// TwinCAT 3 PLC project TcoIoTests
// Title: TcoIoTests
// Company: Vortex.Library
// ProjectVersion: 1.19.1.1780
// ProgramVersion: 3.1.4024.12
// libraries:
//   Tc2_Standard, * (Beckhoff Automation GmbH)
//   Tc2_System, * (Beckhoff Automation GmbH)
//   Tc3_Module, * (Beckhoff Automation GmbH)
//   TcoCore, 0.6.0.913 (Vortex.Library)
//   TcoIo, 0.6.0.913 (Vortex.Library)
// project tree:
//   / PlcTask.TcTTO
//   POUs/ MAIN.TcPOU, tcc.TcPOU, TestEcatComponent.TcPOU
//   DUTs/IO/PdoEntries/ Status_3D84275F.TcDUT, Ctrl_1EFB4D3B.TcDUT, Ctrl_71604E86.TcDUT, Status_B0753356.TcDUT, Status_F2CE6D91.TcDUT, U1_Status_DC903920.TcDUT, U1_Samples_25492287.TcDUT, I1_Status_DC903920.TcDUT, I1_Samples_25492287.TcDUT, U2_Status_DC903920.TcDUT, U2_Samples_25492287.TcDUT, I2_Status_DC903920.TcDUT, I2_Samples_25492287.TcDUT, U3_Status_DC903920.TcDUT, U3_Samples_25492287.TcDUT, I3_Status_DC903920.TcDUT, I3_Samples_25492287.TcDUT, StartTimeNextLatch_02E0C1C8.TcDUT, Status_642C2ED1.TcDUT, Ctrl_77460BD3.TcDUT, Outputs_A910484D.TcDUT, Status_B6795845.TcDUT, Control_C948E0F2.TcDUT, Status_439F40C3.TcDUT, Settings_24C04940.TcDUT, Control_E49DBA1B.TcDUT, Status_8CBE219F.TcDUT, Control_6EF2C5D0.TcDUT
//   DUTs/IO/PDOs/ COM_TxPDO_Map_Inputs_Channel_3801C95E.TcDUT, COM_RxPDO_Map_Outputs_Channel_EADA2E0D.TcDUT, Channel_830843C1.TcDUT, Channel_42CA91F7.TcDUT, AO_Output_Channel_BA7EBB7C.TcDUT, COM_Inputs_3801C95E.TcDUT, COM_Outputs_DEF408EC.TcDUT, AI_Standard_Channel_A8DF64E3.TcDUT, AI_Standard_Channel_4A394481.TcDUT, L1_Voltage_Status_7371B043.TcDUT, L1_Voltage_Samples_41AEB7FF.TcDUT, L1_Current_Status_82DECBF6.TcDUT, L1_Current_Samples_9EC08B3E.TcDUT, L2_Voltage_Status_0D1813FE.TcDUT, L2_Voltage_Samples_75D833AF.TcDUT, L2_Current_Status_FCB7684B.TcDUT, L2_Current_Samples_AAB60F6E.TcDUT, L3_Voltage_Status_273F7295.TcDUT, L3_Voltage_Samples_660A4F9F.TcDUT, L3_Current_Status_D6900920.TcDUT, L3_Current_Samples_B964735E.TcDUT, AI_NextSync1Time_6DC4D296.TcDUT, AI_Sample_Count_EA88CAD9.TcDUT, InfoData_B84DBEC5.TcDUT, MTO_Inputs_Channel_53C09E8B.TcDUT, MTO_Outputs_10x_Channel_A3C0C022.TcDUT, PM_Inputs_Channel_2F868086.TcDUT, PM_Status_data_2A9514CB.TcDUT, PM_Outputs_Channel_E5FBDE30.TcDUT, AT_x_4EC2E768.TcDUT, MDT_864618EC.TcDUT, InfoData_F60A43AC.TcDUT, Device_State_B9CC7757.TcDUT, Device_Control_33EFE70E.TcDUT, Inputs_03C60166.TcDUT, Outputs_79BC345B.TcDUT, Module_1_32_Byte_Valve_Unit_0x7F_1A3DA03C.TcDUT, InfoData_8F85596B.TcDUT, Device_State_384275F8.TcDUT, Device_Control_5857DF0F.TcDUT, Inputs_23559BB0.TcDUT, Outputs_FC2FACAD.TcDUT, Module_1_32_Byte_Valve_Unit_0x7F_85784B27.TcDUT, DI_TxPDO_Map_DF955083.TcDUT, DO_RxPDO_Map_8BCFF4C9.TcDUT, DCM_Status_Channel_36ED096F.TcDUT, DCM_Synchron_info_data_Channel_6FB37C88.TcDUT, DCM_Control_Channel_5A8B5016.TcDUT, DCM_Velocity_Channel_A47A3F41.TcDUT, InfoData_F38373C9.TcDUT, Inputs_424E3ECB.TcDUT, Inputs_84513182.TcDUT, Outputs_3179CEF4.TcDUT, NewMessageFlag_557A079F.TcDUT, Gateway_to_EtherCAT_Data_100_Bytes_AE1F4D6F.TcDUT, EtherCAT_to_Gateway_Data_100_Bytes_44CA1D22.TcDUT, FB_Position_3FA094ED.TcDUT, DRV_Statusword_9B36FDFC.TcDUT, DRV_Following_error_actual_value_5AA320BF.TcDUT, DRV_Controlword_F3F14721.TcDUT, DRV_Target_position_05240F14.TcDUT, InfoData_433F0777.TcDUT, SAI_Inputs_Channel_9DCD6557.TcDUT, SAI_Range_Channel_BDBF6DA9.TcDUT, SAI_Inputs_Real_Channel_CCECF13D.TcDUT, SAI_Range_Control_Channel_F5D9BC22.TcDUT, In_389F2F15.TcDUT, Out_81AAEF2D.TcDUT, ENC_Status_compact_4D066E1A.TcDUT, STM_Status_36ED096F.TcDUT, ENC_Control_compact_21E2D14D.TcDUT, STM_Control_5A8B5016.TcDUT, STM_Velocity_A47A3F41.TcDUT, InfoData_D50C8545.TcDUT, AT_x_26CC547D.TcDUT
//   DUTs/IO/Boxes/ EK1200_013D0B49.TcDUT, EL6002_CD897635.TcDUT, EL1809_32157CFD.TcDUT, EL2809_2B6483BD.TcDUT, EL4004_E203F875.TcDUT, EL6001_0DE01E7E.TcDUT, EL9011_D65D3D32.TcDUT, EK1100_1FC0878B.TcDUT, EK1122_1FC0878B.TcDUT, EL3174_B71BFF42.TcDUT, EL3011_7A495228.TcDUT, EL2008_E2806B95.TcDUT, EK1110_1FC0878B.TcDUT, EL1819_32157CFD.TcDUT, EL2788_E2806B95.TcDUT, EL3773_F128CC82.TcDUT, EL2258_E3B260FA.TcDUT, EL3164_B71BFF42.TcDUT, EL3403_812980A6.TcDUT, EL3024_C6E76B5A.TcDUT, AX5101_1BD22F51.TcDUT, AX5106_1BD22F51.TcDUT, AES_A3B07071.TcDUT, EL6631_A0EC075C.TcDUT, EL9010_D29C2085.TcDUT, AES_B47A2610.TcDUT, IMecat_x_75C6CB6B.TcDUT, AX5103_1BD22F51.TcDUT, EL7332_DFB2BED7.TcDUT, CMMP_93B92D52.TcDUT, Flexi_Gateway_GETC1_429ECB70.TcDUT, EL7211_008D5C9A.TcDUT, EL3692_73B94100.TcDUT, EPP1322_1FC0878B.TcDUT, EPP1008_78E8D3DD.TcDUT, EPP1332_1FC0878B.TcDUT, Flexi_Soft_EtherCAT_Gateway_DE394EDD.TcDUT, EL7041_86DE63E7.TcDUT, IndraDrive_MPB20_C66205C3.TcDUT, EPP2308_F6D9A8D1.TcDUT
//   DUTs/IO/Devices/ SyncUnitTasks_5FDC9770.TcDUT, SyncUnits_C3A34B50.TcDUT, SyncUnits_F0D163CC.TcDUT, SyncUnits_5BE71B8B.TcDUT
//   DUTs/IO/Topology/ Term_1_EK1200_B38DC9A8.TcDUT, Device_1_EtherCAT_49C09C66.TcDUT, Term_11_EK1100_B6553301.TcDUT, Term_18_EK1100_20659A8D.TcDUT, Term_25_EK1100_08217EB4.TcDUT, Term_28_EK1100_415F4A7E.TcDUT, Term_24_EK1122_39E7B5CB.TcDUT, Term_23_EK1100_DFBF0BE4.TcDUT, Term_10_EK1122_3D069EC1.TcDUT, Term_9_EK1100_91BFEC25.TcDUT, Device_2_EtherCAT_22CD061B.TcDUT, Term_157_EK1100_7C4BDD77.TcDUT, Term_158_EK1100_E3D699B1.TcDUT, Term_154_EK1122_E57516AE.TcDUT, Term_153_EK1100_91C0BB48.TcDUT, Term_180_EK1100_796B7783.TcDUT, Term_182_EK1100_E6B2C35E.TcDUT, Term_179_EK1122_2A33725A.TcDUT, Term_178_EK1100_9B7E9852.TcDUT, Term_147_EK1122_CA6A5D16.TcDUT, Term_189_EK1100_06A16014.TcDUT, Term_194_EK1100_D4E2C05F.TcDUT, Term_188_EK1122_78D8AA43.TcDUT, Term_187_EK1100_648C31BD.TcDUT, Term_231_EK1100_6FCE8CEB.TcDUT, Term_233_EK1100_CB654C3B.TcDUT, Term_230_EK1122_16418046.TcDUT, Term_207_EK1100_2D36550A.TcDUT, Term_186_EK1122_75C79D52.TcDUT, Term_237_EK1122_86A8F7BD.TcDUT, Term_289_EK1100_9C677E50.TcDUT, Term_294_EK1100_DFE2A59E.TcDUT, Term_331_EK1100_B9C4E092.TcDUT, Term_333_EK1100_1D6F2042.TcDUT, Term_330_EK1122_0EDE60FE.TcDUT, Term_307_EK1100_EB8FAA41.TcDUT, Term_288_EK1122_18F8921F.TcDUT, Term_146_EK1100_439F5464.TcDUT, Device_3_EtherCAT_368E547E.TcDUT, R1_A2_EC_EK1122_F4361AFD.TcDUT, R1_A3_EC_EK1122_981C12E1.TcDUT, R1_A4_X1_EK1100_C601B400.TcDUT, R1_A4_X2_A2_EK1122_39ABCC27.TcDUT, R1_A4_X2_EK1100_6F5FB3BA.TcDUT, R1_A4_EC_EK1122_467C5A0B.TcDUT, R1_EK1100_4AD22B7B.TcDUT, R2_A2_EC_EK1122_6D3594D4.TcDUT, R2_EK1100_10D8A594.TcDUT, R3_A2_EC_EK1122_9D59CDC8.TcDUT, R3_EK1100_C7887D6C.TcDUT, RH_A2_X2_EK1100_67419BB1.TcDUT, RH_A2_EK1122_10728E09.TcDUT, RH_EK1100_A5940DFE.TcDUT, R4_A2_EC_EK1122_254454A1.TcDUT, R4_EK1100_46A1248C.TcDUT, A2_EK1122_967E4A9C.TcDUT, R4A_EK1100_48316913.TcDUT, R5_A2_EC_EK1122_D562526C.TcDUT, R5_EK1100_0007A337.TcDUT, R6_EK1100_8C41F5F2.TcDUT, R7_A2_EC_EK1122_B7F046E4.TcDUT, R7_EK1100_F50DDAC8.TcDUT, R8_AB0_EPP1322_0001_1BB6BCA8.TcDUT, R8_A2_EK1122_E74C4B62.TcDUT, R8_A3_EK1122_71CA94BA.TcDUT, RC10_A2_EK1122_BBB6F36B.TcDUT, RC10_EPP_EPP1322_0001_810E0540.TcDUT, RC10_A3_EK1122_A50FC1ED.TcDUT, RC10_1_EK1100_40BAEC0F.TcDUT, RC10_2_EK1100_27865421.TcDUT, RC20_A2_EK1122_77321D67.TcDUT, RC20_EPP_EPP1322_0001_59D450BA.TcDUT, RC20_A3_EK1122_1263CE61.TcDUT, RC20_1_EK1100_F221D0A9.TcDUT, RC20_2_EK1100_5EABB509.TcDUT, R8_A8_EK1122_2533F93A.TcDUT, RC30_A2_EK1122_334E4763.TcDUT, RC30_EPP_EPP1322_0001_EDDD6881.TcDUT, RC30_A3_EK1122_482A08F6.TcDUT, RC30_1_EK1100_B995809E.TcDUT, RC30_2_EK1100_8A0FE17C.TcDUT, RC40_A2_EK1122_EAFADCC8.TcDUT, RC40_EPP_EPP1322_0001_ECA1E6F9.TcDUT, RC40_A3_EK1122_E505EE87.TcDUT, RC40_1_EK1100_B918F64D.TcDUT, RC40_2_EK1100_ACF07759.TcDUT, R8_A9_EK1122_3EDD8752.TcDUT, RC50_A2_EK1122_AE8686CC.TcDUT, RC50_EPP_EPP1322_0001_58A8DEC2.TcDUT, RC50_A3_EK1122_7F1D927D.TcDUT, RC50_1_EK1100_D6E64946.TcDUT, RC50_2_EK1100_7854232C.TcDUT, RC60_A2_EK1122_620268C0.TcDUT, RC60_EPP_EPP1322_0001_80728B38.TcDUT, RC60_A3_EK1122_0BEA55B5.TcDUT, RC60_1_EK1100_9BABA6E0.TcDUT, RC60_2_EK1100_0179C204.TcDUT, R8_A10_EK1122_484442E0.TcDUT, RC70_A2_EK1122_267E32C4.TcDUT, RC70_EPP_EPP1322_0001_347BB303.TcDUT, RC70_A3_EK1122_27C9256F.TcDUT, RC70_1_EK1100_B905944A.TcDUT, RC70_2_EK1100_D5DD9671.TcDUT, RC80_A2_EK1122_C3467012.TcDUT, RC80_EPP_EPP1322_0001_828B97C8.TcDUT, RC80_A3_EK1122_B1484BA9.TcDUT, RC80_1_EK1100_5DD08FF5.TcDUT, RC80_2_EK1100_DC1461B5.TcDUT, R8_A11_EK1122_3ED7E2A8.TcDUT, RP10_A2_EK1122_55AC9C5A.TcDUT, RP10_EK1100_26DB4001.TcDUT, RP20_A2_EK1122_68D808EA.TcDUT, RP20_EK1100_7A23D5FF.TcDUT, R8_A12_EK1122_5B843125.TcDUT, RP30_A2_EK1122_C3CC9CB4.TcDUT, RP30_EK1100_66AE6AB6.TcDUT, R8_A13_EK1122_C6957FFB.TcDUT, R8_EK1100_9C7B3B67.TcDUT, R9_AB0_EPP1322_0001_BD7A28FA.TcDUT, R9_A2_EK1122_81F50509.TcDUT, R9_A3_EK1122_C18C26F5.TcDUT, R9_EK1100_484053C0.TcDUT, R10_A2_EK1122_75D61001.TcDUT, R10_AB01_EPP1332_0001_D97A7767.TcDUT, R10_AB00_EPP1322_0001_481BC624.TcDUT, R10_A3_EK1122_6A26DC25.TcDUT, R10_EK1100_C5CE1D87.TcDUT, Device_4_EtherCAT_07442C6B.TcDUT, Term_279_EK1100_ED7D6272.TcDUT, Term_554_EK1100_B580E218.TcDUT, Term_748_EK1100_BC4343B1.TcDUT, Term_881_EK1100_F732F370.TcDUT, Term_1047_EK1100_7ACEE53D.TcDUT, Device_5_EtherCAT_0A694E3C.TcDUT
//   GVLs/ GVL_iXlinker.TcGVL
// (motion and I/O tree: see PLC project tcoio)
// real-time tasks:
//   TASK PlcTask: cycle T#10ms, priority 20, ADS port 350
//   TASK PlcTask1: cycle T#10ms, priority 21, ADS port 351
//   TASK PlcTask2: cycle T#10ms, priority 22, ADS port 352
// variable links:
//   TcoIoTests/TcoIoTests Instance <-> Device 1 (EtherCAT)
//     PlcTask Inputs/GVL_iXlinker.Device_1_EtherCAT.InfoData.AmsNetId <-> InfoData/AmsNetId
//     PlcTask Inputs/GVL_iXlinker.Device_1_EtherCAT.InfoData.CfgSlaveCount <-> InfoData/CfgSlaveCount
//     PlcTask Inputs/GVL_iXlinker.Device_1_EtherCAT.InfoData.ChangeCount <-> InfoData/ChangeCount
//     PlcTask Inputs/GVL_iXlinker.Device_1_EtherCAT.InfoData.DevId <-> InfoData/DevId
//     PlcTask Inputs/GVL_iXlinker.Device_1_EtherCAT.Inputs.DevState <-> Inputs/DevState
//     PlcTask Inputs/GVL_iXlinker.Device_1_EtherCAT.Inputs.Frm0InputToggle <-> Inputs/Frm0InputToggle
//     PlcTask Inputs/GVL_iXlinker.Device_1_EtherCAT.Inputs.Frm0State <-> Inputs/Frm0State
//     PlcTask Inputs/GVL_iXlinker.Device_1_EtherCAT.Inputs.Frm0WcState <-> Inputs/Frm0WcState
//     PlcTask Inputs/GVL_iXlinker.Device_1_EtherCAT.Inputs.SlaveCount <-> Inputs/SlaveCount
//     PlcTask Inputs/GVL_iXlinker.Device_1_EtherCAT.SyncUnits._default.PlcTask1.InfoData.ObjectId <-> SyncUnits/<default>/PlcTask1/InfoData/ObjectId
//     PlcTask Inputs/GVL_iXlinker.Device_1_EtherCAT.SyncUnits._default.PlcTask1.InfoData.SlaveCount <-> SyncUnits/<default>/PlcTask1/InfoData/SlaveCount
//     PlcTask Inputs/GVL_iXlinker.Device_1_EtherCAT.SyncUnits._default.PlcTask1.InfoData.State <-> SyncUnits/<default>/PlcTask1/InfoData/State
//     PlcTask Inputs/GVL_iXlinker.Device_1_EtherCAT.SyncUnits._default.PlcTask1.WcState.WcState <-> SyncUnits/<default>/PlcTask1/WcState/WcState
//     PlcTask Outputs/GVL_iXlinker.Device_1_EtherCAT.Outputs.DevCtrl <-> Outputs/DevCtrl
//     PlcTask Outputs/GVL_iXlinker.Device_1_EtherCAT.Outputs.Frm0Ctrl <-> Outputs/Frm0Ctrl
//     PlcTask Outputs/GVL_iXlinker.Device_1_EtherCAT.Outputs.Frm0WcCtrl <-> Outputs/Frm0WcCtrl
//   TcoIoTests/TcoIoTests Instance <-> Device 1 (EtherCAT)/Term 1 (EK1200)/Term 2 (EL6002)
//     PlcTask Inputs/GVL_iXlinker.Device_1_EtherCAT.Term_1_EK1200.Term_2_EL6002.COM_TxPDO_Map_Inputs_Channel_1.Data_In[0] <-> COM TxPDO-Map Inputs Channel 1/Data In 0
//     PlcTask Inputs/GVL_iXlinker.Device_1_EtherCAT.Term_1_EK1200.Term_2_EL6002.COM_TxPDO_Map_Inputs_Channel_1.Data_In[10] <-> COM TxPDO-Map Inputs Channel 1/Data In 10
//     PlcTask Inputs/GVL_iXlinker.Device_1_EtherCAT.Term_1_EK1200.Term_2_EL6002.COM_TxPDO_Map_Inputs_Channel_1.Data_In[11] <-> COM TxPDO-Map Inputs Channel 1/Data In 11
//     PlcTask Inputs/GVL_iXlinker.Device_1_EtherCAT.Term_1_EK1200.Term_2_EL6002.COM_TxPDO_Map_Inputs_Channel_1.Data_In[12] <-> COM TxPDO-Map Inputs Channel 1/Data In 12
//     PlcTask Inputs/GVL_iXlinker.Device_1_EtherCAT.Term_1_EK1200.Term_2_EL6002.COM_TxPDO_Map_Inputs_Channel_1.Data_In[13] <-> COM TxPDO-Map Inputs Channel 1/Data In 13
//     PlcTask Inputs/GVL_iXlinker.Device_1_EtherCAT.Term_1_EK1200.Term_2_EL6002.COM_TxPDO_Map_Inputs_Channel_1.Data_In[14] <-> COM TxPDO-Map Inputs Channel 1/Data In 14
//     PlcTask Inputs/GVL_iXlinker.Device_1_EtherCAT.Term_1_EK1200.Term_2_EL6002.COM_TxPDO_Map_Inputs_Channel_1.Data_In[15] <-> COM TxPDO-Map Inputs Channel 1/Data In 15
//     PlcTask Inputs/GVL_iXlinker.Device_1_EtherCAT.Term_1_EK1200.Term_2_EL6002.COM_TxPDO_Map_Inputs_Channel_1.Data_In[16] <-> COM TxPDO-Map Inputs Channel 1/Data In 16
//     PlcTask Inputs/GVL_iXlinker.Device_1_EtherCAT.Term_1_EK1200.Term_2_EL6002.COM_TxPDO_Map_Inputs_Channel_1.Data_In[17] <-> COM TxPDO-Map Inputs Channel 1/Data In 17
//     PlcTask Inputs/GVL_iXlinker.Device_1_EtherCAT.Term_1_EK1200.Term_2_EL6002.COM_TxPDO_Map_Inputs_Channel_1.Data_In[18] <-> COM TxPDO-Map Inputs Channel 1/Data In 18
//     PlcTask Inputs/GVL_iXlinker.Device_1_EtherCAT.Term_1_EK1200.Term_2_EL6002.COM_TxPDO_Map_Inputs_Channel_1.Data_In[19] <-> COM TxPDO-Map Inputs Channel 1/Data In 19
//     PlcTask Inputs/GVL_iXlinker.Device_1_EtherCAT.Term_1_EK1200.Term_2_EL6002.COM_TxPDO_Map_Inputs_Channel_1.Data_In[1] <-> COM TxPDO-Map Inputs Channel 1/Data In 1
//     PlcTask Inputs/GVL_iXlinker.Device_1_EtherCAT.Term_1_EK1200.Term_2_EL6002.COM_TxPDO_Map_Inputs_Channel_1.Data_In[20] <-> COM TxPDO-Map Inputs Channel 1/Data In 20
//     PlcTask Inputs/GVL_iXlinker.Device_1_EtherCAT.Term_1_EK1200.Term_2_EL6002.COM_TxPDO_Map_Inputs_Channel_1.Data_In[21] <-> COM TxPDO-Map Inputs Channel 1/Data In 21
//     PlcTask Inputs/GVL_iXlinker.Device_1_EtherCAT.Term_1_EK1200.Term_2_EL6002.COM_TxPDO_Map_Inputs_Channel_1.Data_In[2] <-> COM TxPDO-Map Inputs Channel 1/Data In 2
//     PlcTask Inputs/GVL_iXlinker.Device_1_EtherCAT.Term_1_EK1200.Term_2_EL6002.COM_TxPDO_Map_Inputs_Channel_1.Data_In[3] <-> COM TxPDO-Map Inputs Channel 1/Data In 3
//     PlcTask Inputs/GVL_iXlinker.Device_1_EtherCAT.Term_1_EK1200.Term_2_EL6002.COM_TxPDO_Map_Inputs_Channel_1.Data_In[4] <-> COM TxPDO-Map Inputs Channel 1/Data In 4
//     PlcTask Inputs/GVL_iXlinker.Device_1_EtherCAT.Term_1_EK1200.Term_2_EL6002.COM_TxPDO_Map_Inputs_Channel_1.Data_In[5] <-> COM TxPDO-Map Inputs Channel 1/Data In 5
//     PlcTask Inputs/GVL_iXlinker.Device_1_EtherCAT.Term_1_EK1200.Term_2_EL6002.COM_TxPDO_Map_Inputs_Channel_1.Data_In[6] <-> COM TxPDO-Map Inputs Channel 1/Data In 6
//     PlcTask Inputs/GVL_iXlinker.Device_1_EtherCAT.Term_1_EK1200.Term_2_EL6002.COM_TxPDO_Map_Inputs_Channel_1.Data_In[7] <-> COM TxPDO-Map Inputs Channel 1/Data In 7
//     PlcTask Inputs/GVL_iXlinker.Device_1_EtherCAT.Term_1_EK1200.Term_2_EL6002.COM_TxPDO_Map_Inputs_Channel_1.Data_In[8] <-> COM TxPDO-Map Inputs Channel 1/Data In 8
//     PlcTask Inputs/GVL_iXlinker.Device_1_EtherCAT.Term_1_EK1200.Term_2_EL6002.COM_TxPDO_Map_Inputs_Channel_1.Data_In[9] <-> COM TxPDO-Map Inputs Channel 1/Data In 9
//     PlcTask Inputs/GVL_iXlinker.Device_1_EtherCAT.Term_1_EK1200.Term_2_EL6002.COM_TxPDO_Map_Inputs_Channel_2.Data_In[0] <-> COM TxPDO-Map Inputs Channel 2/Data In 0
//     PlcTask Inputs/GVL_iXlinker.Device_1_EtherCAT.Term_1_EK1200.Term_2_EL6002.COM_TxPDO_Map_Inputs_Channel_2.Data_In[10] <-> COM TxPDO-Map Inputs Channel 2/Data In 10
//     PlcTask Inputs/GVL_iXlinker.Device_1_EtherCAT.Term_1_EK1200.Term_2_EL6002.COM_TxPDO_Map_Inputs_Channel_2.Data_In[11] <-> COM TxPDO-Map Inputs Channel 2/Data In 11
//     PlcTask Inputs/GVL_iXlinker.Device_1_EtherCAT.Term_1_EK1200.Term_2_EL6002.COM_TxPDO_Map_Inputs_Channel_2.Data_In[12] <-> COM TxPDO-Map Inputs Channel 2/Data In 12
//     PlcTask Inputs/GVL_iXlinker.Device_1_EtherCAT.Term_1_EK1200.Term_2_EL6002.COM_TxPDO_Map_Inputs_Channel_2.Data_In[13] <-> COM TxPDO-Map Inputs Channel 2/Data In 13
//     PlcTask Inputs/GVL_iXlinker.Device_1_EtherCAT.Term_1_EK1200.Term_2_EL6002.COM_TxPDO_Map_Inputs_Channel_2.Data_In[14] <-> COM TxPDO-Map Inputs Channel 2/Data In 14
//     PlcTask Inputs/GVL_iXlinker.Device_1_EtherCAT.Term_1_EK1200.Term_2_EL6002.COM_TxPDO_Map_Inputs_Channel_2.Data_In[15] <-> COM TxPDO-Map Inputs Channel 2/Data In 15
//     PlcTask Inputs/GVL_iXlinker.Device_1_EtherCAT.Term_1_EK1200.Term_2_EL6002.COM_TxPDO_Map_Inputs_Channel_2.Data_In[16] <-> COM TxPDO-Map Inputs Channel 2/Data In 16
//     PlcTask Inputs/GVL_iXlinker.Device_1_EtherCAT.Term_1_EK1200.Term_2_EL6002.COM_TxPDO_Map_Inputs_Channel_2.Data_In[17] <-> COM TxPDO-Map Inputs Channel 2/Data In 17
//     PlcTask Inputs/GVL_iXlinker.Device_1_EtherCAT.Term_1_EK1200.Term_2_EL6002.COM_TxPDO_Map_Inputs_Channel_2.Data_In[18] <-> COM TxPDO-Map Inputs Channel 2/Data In 18
//     PlcTask Inputs/GVL_iXlinker.Device_1_EtherCAT.Term_1_EK1200.Term_2_EL6002.COM_TxPDO_Map_Inputs_Channel_2.Data_In[19] <-> COM TxPDO-Map Inputs Channel 2/Data In 19
//     PlcTask Inputs/GVL_iXlinker.Device_1_EtherCAT.Term_1_EK1200.Term_2_EL6002.COM_TxPDO_Map_Inputs_Channel_2.Data_In[1] <-> COM TxPDO-Map Inputs Channel 2/Data In 1
//     PlcTask Inputs/GVL_iXlinker.Device_1_EtherCAT.Term_1_EK1200.Term_2_EL6002.COM_TxPDO_Map_Inputs_Channel_2.Data_In[20] <-> COM TxPDO-Map Inputs Channel 2/Data In 20
//     PlcTask Inputs/GVL_iXlinker.Device_1_EtherCAT.Term_1_EK1200.Term_2_EL6002.COM_TxPDO_Map_Inputs_Channel_2.Data_In[21] <-> COM TxPDO-Map Inputs Channel 2/Data In 21
//     PlcTask Inputs/GVL_iXlinker.Device_1_EtherCAT.Term_1_EK1200.Term_2_EL6002.COM_TxPDO_Map_Inputs_Channel_2.Data_In[2] <-> COM TxPDO-Map Inputs Channel 2/Data In 2
//     PlcTask Inputs/GVL_iXlinker.Device_1_EtherCAT.Term_1_EK1200.Term_2_EL6002.COM_TxPDO_Map_Inputs_Channel_2.Data_In[3] <-> COM TxPDO-Map Inputs Channel 2/Data In 3
//     PlcTask Inputs/GVL_iXlinker.Device_1_EtherCAT.Term_1_EK1200.Term_2_EL6002.COM_TxPDO_Map_Inputs_Channel_2.Data_In[4] <-> COM TxPDO-Map Inputs Channel 2/Data In 4
//     PlcTask Inputs/GVL_iXlinker.Device_1_EtherCAT.Term_1_EK1200.Term_2_EL6002.COM_TxPDO_Map_Inputs_Channel_2.Data_In[5] <-> COM TxPDO-Map Inputs Channel 2/Data In 5
//     PlcTask Inputs/GVL_iXlinker.Device_1_EtherCAT.Term_1_EK1200.Term_2_EL6002.COM_TxPDO_Map_Inputs_Channel_2.Data_In[6] <-> COM TxPDO-Map Inputs Channel 2/Data In 6
//     PlcTask Inputs/GVL_iXlinker.Device_1_EtherCAT.Term_1_EK1200.Term_2_EL6002.COM_TxPDO_Map_Inputs_Channel_2.Data_In[7] <-> COM TxPDO-Map Inputs Channel 2/Data In 7
//     PlcTask Inputs/GVL_iXlinker.Device_1_EtherCAT.Term_1_EK1200.Term_2_EL6002.COM_TxPDO_Map_Inputs_Channel_2.Data_In[8] <-> COM TxPDO-Map Inputs Channel 2/Data In 8
//     PlcTask Inputs/GVL_iXlinker.Device_1_EtherCAT.Term_1_EK1200.Term_2_EL6002.COM_TxPDO_Map_Inputs_Channel_2.Data_In[9] <-> COM TxPDO-Map Inputs Channel 2/Data In 9
//     PlcTask Inputs/GVL_iXlinker.Device_1_EtherCAT.Term_1_EK1200.Term_2_EL6002.COM_TxPDO_Map_Inputs_Channel_1.Status/Buffer_full <-> COM TxPDO-Map Inputs Channel 1/Status/Buffer full
//     PlcTask Inputs/GVL_iXlinker.Device_1_EtherCAT.Term_1_EK1200.Term_2_EL6002.COM_TxPDO_Map_Inputs_Channel_2.Status/Buffer_full <-> COM TxPDO-Map Inputs Channel 2/Status/Buffer full
//     PlcTask Inputs/GVL_iXlinker.Device_1_EtherCAT.Term_1_EK1200.Term_2_EL6002.COM_TxPDO_Map_Inputs_Channel_1.Status/Framing_error <-> COM TxPDO-Map Inputs Channel 1/Status/Framing error
//     PlcTask Inputs/GVL_iXlinker.Device_1_EtherCAT.Term_1_EK1200.Term_2_EL6002.COM_TxPDO_Map_Inputs_Channel_2.Status/Framing_error <-> COM TxPDO-Map Inputs Channel 2/Status/Framing error
//     PlcTask Inputs/GVL_iXlinker.Device_1_EtherCAT.Term_1_EK1200.Term_2_EL6002.COM_TxPDO_Map_Inputs_Channel_1.Status/Init_accepted <-> COM TxPDO-Map Inputs Channel 1/Status/Init accepted
//     PlcTask Inputs/GVL_iXlinker.Device_1_EtherCAT.Term_1_EK1200.Term_2_EL6002.COM_TxPDO_Map_Inputs_Channel_2.Status/Init_accepted <-> COM TxPDO-Map Inputs Channel 2/Status/Init accepted
//     PlcTask Inputs/GVL_iXlinker.Device_1_EtherCAT.Term_1_EK1200.Term_2_EL6002.COM_TxPDO_Map_Inputs_Channel_1.Status/Input_length <-> COM TxPDO-Map Inputs Channel 1/Status/Input length
//     PlcTask Inputs/GVL_iXlinker.Device_1_EtherCAT.Term_1_EK1200.Term_2_EL6002.COM_TxPDO_Map_Inputs_Channel_2.Status/Input_length <-> COM TxPDO-Map Inputs Channel 2/Status/Input length
//     PlcTask Inputs/GVL_iXlinker.Device_1_EtherCAT.Term_1_EK1200.Term_2_EL6002.COM_TxPDO_Map_Inputs_Channel_1.Status/Overrun_error <-> COM TxPDO-Map Inputs Channel 1/Status/Overrun error
//     PlcTask Inputs/GVL_iXlinker.Device_1_EtherCAT.Term_1_EK1200.Term_2_EL6002.COM_TxPDO_Map_Inputs_Channel_2.Status/Overrun_error <-> COM TxPDO-Map Inputs Channel 2/Status/Overrun error
//     PlcTask Inputs/GVL_iXlinker.Device_1_EtherCAT.Term_1_EK1200.Term_2_EL6002.COM_TxPDO_Map_Inputs_Channel_1.Status/Parity_error <-> COM TxPDO-Map Inputs Channel 1/Status/Parity error
//     PlcTask Inputs/GVL_iXlinker.Device_1_EtherCAT.Term_1_EK1200.Term_2_EL6002.COM_TxPDO_Map_Inputs_Channel_2.Status/Parity_error <-> COM TxPDO-Map Inputs Channel 2/Status/Parity error
//     PlcTask Inputs/GVL_iXlinker.Device_1_EtherCAT.Term_1_EK1200.Term_2_EL6002.COM_TxPDO_Map_Inputs_Channel_1.Status/Receive_request <-> COM TxPDO-Map Inputs Channel 1/Status/Receive request
//     PlcTask Inputs/GVL_iXlinker.Device_1_EtherCAT.Term_1_EK1200.Term_2_EL6002.COM_TxPDO_Map_Inputs_Channel_2.Status/Receive_request <-> COM TxPDO-Map Inputs Channel 2/Status/Receive request
//     PlcTask Inputs/GVL_iXlinker.Device_1_EtherCAT.Term_1_EK1200.Term_2_EL6002.COM_TxPDO_Map_Inputs_Channel_1.Status/Transmit_accepted <-> COM TxPDO-Map Inputs Channel 1/Status/Transmit accepted
//     PlcTask Inputs/GVL_iXlinker.Device_1_EtherCAT.Term_1_EK1200.Term_2_EL6002.COM_TxPDO_Map_Inputs_Channel_2.Status/Transmit_accepted <-> COM TxPDO-Map Inputs Channel 2/Status/Transmit accepted
//     PlcTask Inputs/GVL_iXlinker.Device_1_EtherCAT.Term_1_EK1200.Term_2_EL6002.InfoData.AdsAddr <-> InfoData/AdsAddr
//     PlcTask Inputs/GVL_iXlinker.Device_1_EtherCAT.Term_1_EK1200.Term_2_EL6002.InfoData.State <-> InfoData/State
//     PlcTask Inputs/GVL_iXlinker.Device_1_EtherCAT.Term_1_EK1200.Term_2_EL6002.WcState.InputToggle <-> WcState/InputToggle
//     PlcTask Inputs/GVL_iXlinker.Device_1_EtherCAT.Term_1_EK1200.Term_2_EL6002.WcState.WcState <-> WcState/WcState
//     PlcTask Outputs/GVL_iXlinker.Device_1_EtherCAT.Term_1_EK1200.Term_2_EL6002.COM_RxPDO_Map_Outputs_Channel_1.Ctrl/Init_request <-> COM RxPDO-Map Outputs Channel 1/Ctrl/Init request
//     PlcTask Outputs/GVL_iXlinker.Device_1_EtherCAT.Term_1_EK1200.Term_2_EL6002.COM_RxPDO_Map_Outputs_Channel_2.Ctrl/Init_request <-> COM RxPDO-Map Outputs Channel 2/Ctrl/Init request
//     PlcTask Outputs/GVL_iXlinker.Device_1_EtherCAT.Term_1_EK1200.Term_2_EL6002.COM_RxPDO_Map_Outputs_Channel_1.Ctrl/Output_length <-> COM RxPDO-Map Outputs Channel 1/Ctrl/Output length
//     PlcTask Outputs/GVL_iXlinker.Device_1_EtherCAT.Term_1_EK1200.Term_2_EL6002.COM_RxPDO_Map_Outputs_Channel_2.Ctrl/Output_length <-> COM RxPDO-Map Outputs Channel 2/Ctrl/Output length
//     PlcTask Outputs/GVL_iXlinker.Device_1_EtherCAT.Term_1_EK1200.Term_2_EL6002.COM_RxPDO_Map_Outputs_Channel_1.Ctrl/Receive_accepted <-> COM RxPDO-Map Outputs Channel 1/Ctrl/Receive accepted
//     PlcTask Outputs/GVL_iXlinker.Device_1_EtherCAT.Term_1_EK1200.Term_2_EL6002.COM_RxPDO_Map_Outputs_Channel_2.Ctrl/Receive_accepted <-> COM RxPDO-Map Outputs Channel 2/Ctrl/Receive accepted
//     PlcTask Outputs/GVL_iXlinker.Device_1_EtherCAT.Term_1_EK1200.Term_2_EL6002.COM_RxPDO_Map_Outputs_Channel_1.Ctrl/Send_continuous <-> COM RxPDO-Map Outputs Channel 1/Ctrl/Send continuous
//     PlcTask Outputs/GVL_iXlinker.Device_1_EtherCAT.Term_1_EK1200.Term_2_EL6002.COM_RxPDO_Map_Outputs_Channel_2.Ctrl/Send_continuous <-> COM RxPDO-Map Outputs Channel 2/Ctrl/Send continuous
//     PlcTask Outputs/GVL_iXlinker.Device_1_EtherCAT.Term_1_EK1200.Term_2_EL6002.COM_RxPDO_Map_Outputs_Channel_1.Ctrl/Transmit_request <-> COM RxPDO-Map Outputs Channel 1/Ctrl/Transmit request
//     PlcTask Outputs/GVL_iXlinker.Device_1_EtherCAT.Term_1_EK1200.Term_2_EL6002.COM_RxPDO_Map_Outputs_Channel_2.Ctrl/Transmit_request <-> COM RxPDO-Map Outputs Channel 2/Ctrl/Transmit request
//     PlcTask Outputs/GVL_iXlinker.Device_1_EtherCAT.Term_1_EK1200.Term_2_EL6002.COM_RxPDO_Map_Outputs_Channel_1.Data_Out[0] <-> COM RxPDO-Map Outputs Channel 1/Data Out 0
//     PlcTask Outputs/GVL_iXlinker.Device_1_EtherCAT.Term_1_EK1200.Term_2_EL6002.COM_RxPDO_Map_Outputs_Channel_1.Data_Out[10] <-> COM RxPDO-Map Outputs Channel 1/Data Out 10
//     PlcTask Outputs/GVL_iXlinker.Device_1_EtherCAT.Term_1_EK1200.Term_2_EL6002.COM_RxPDO_Map_Outputs_Channel_1.Data_Out[11] <-> COM RxPDO-Map Outputs Channel 1/Data Out 11
//     PlcTask Outputs/GVL_iXlinker.Device_1_EtherCAT.Term_1_EK1200.Term_2_EL6002.COM_RxPDO_Map_Outputs_Channel_1.Data_Out[12] <-> COM RxPDO-Map Outputs Channel 1/Data Out 12
//     PlcTask Outputs/GVL_iXlinker.Device_1_EtherCAT.Term_1_EK1200.Term_2_EL6002.COM_RxPDO_Map_Outputs_Channel_1.Data_Out[13] <-> COM RxPDO-Map Outputs Channel 1/Data Out 13
//     PlcTask Outputs/GVL_iXlinker.Device_1_EtherCAT.Term_1_EK1200.Term_2_EL6002.COM_RxPDO_Map_Outputs_Channel_1.Data_Out[14] <-> COM RxPDO-Map Outputs Channel 1/Data Out 14
//     PlcTask Outputs/GVL_iXlinker.Device_1_EtherCAT.Term_1_EK1200.Term_2_EL6002.COM_RxPDO_Map_Outputs_Channel_1.Data_Out[15] <-> COM RxPDO-Map Outputs Channel 1/Data Out 15
//     PlcTask Outputs/GVL_iXlinker.Device_1_EtherCAT.Term_1_EK1200.Term_2_EL6002.COM_RxPDO_Map_Outputs_Channel_1.Data_Out[16] <-> COM RxPDO-Map Outputs Channel 1/Data Out 16
//     PlcTask Outputs/GVL_iXlinker.Device_1_EtherCAT.Term_1_EK1200.Term_2_EL6002.COM_RxPDO_Map_Outputs_Channel_1.Data_Out[17] <-> COM RxPDO-Map Outputs Channel 1/Data Out 17
//     PlcTask Outputs/GVL_iXlinker.Device_1_EtherCAT.Term_1_EK1200.Term_2_EL6002.COM_RxPDO_Map_Outputs_Channel_1.Data_Out[18] <-> COM RxPDO-Map Outputs Channel 1/Data Out 18
//     PlcTask Outputs/GVL_iXlinker.Device_1_EtherCAT.Term_1_EK1200.Term_2_EL6002.COM_RxPDO_Map_Outputs_Channel_1.Data_Out[19] <-> COM RxPDO-Map Outputs Channel 1/Data Out 19
//     PlcTask Outputs/GVL_iXlinker.Device_1_EtherCAT.Term_1_EK1200.Term_2_EL6002.COM_RxPDO_Map_Outputs_Channel_1.Data_Out[1] <-> COM RxPDO-Map Outputs Channel 1/Data Out 1
//     PlcTask Outputs/GVL_iXlinker.Device_1_EtherCAT.Term_1_EK1200.Term_2_EL6002.COM_RxPDO_Map_Outputs_Channel_1.Data_Out[20] <-> COM RxPDO-Map Outputs Channel 1/Data Out 20
//     PlcTask Outputs/GVL_iXlinker.Device_1_EtherCAT.Term_1_EK1200.Term_2_EL6002.COM_RxPDO_Map_Outputs_Channel_1.Data_Out[21] <-> COM RxPDO-Map Outputs Channel 1/Data Out 21
//     PlcTask Outputs/GVL_iXlinker.Device_1_EtherCAT.Term_1_EK1200.Term_2_EL6002.COM_RxPDO_Map_Outputs_Channel_1.Data_Out[2] <-> COM RxPDO-Map Outputs Channel 1/Data Out 2
//     PlcTask Outputs/GVL_iXlinker.Device_1_EtherCAT.Term_1_EK1200.Term_2_EL6002.COM_RxPDO_Map_Outputs_Channel_1.Data_Out[3] <-> COM RxPDO-Map Outputs Channel 1/Data Out 3
//     PlcTask Outputs/GVL_iXlinker.Device_1_EtherCAT.Term_1_EK1200.Term_2_EL6002.COM_RxPDO_Map_Outputs_Channel_1.Data_Out[4] <-> COM RxPDO-Map Outputs Channel 1/Data Out 4
//     PlcTask Outputs/GVL_iXlinker.Device_1_EtherCAT.Term_1_EK1200.Term_2_EL6002.COM_RxPDO_Map_Outputs_Channel_1.Data_Out[5] <-> COM RxPDO-Map Outputs Channel 1/Data Out 5
//     PlcTask Outputs/GVL_iXlinker.Device_1_EtherCAT.Term_1_EK1200.Term_2_EL6002.COM_RxPDO_Map_Outputs_Channel_1.Data_Out[6] <-> COM RxPDO-Map Outputs Channel 1/Data Out 6
//     PlcTask Outputs/GVL_iXlinker.Device_1_EtherCAT.Term_1_EK1200.Term_2_EL6002.COM_RxPDO_Map_Outputs_Channel_1.Data_Out[7] <-> COM RxPDO-Map Outputs Channel 1/Data Out 7
//     PlcTask Outputs/GVL_iXlinker.Device_1_EtherCAT.Term_1_EK1200.Term_2_EL6002.COM_RxPDO_Map_Outputs_Channel_1.Data_Out[8] <-> COM RxPDO-Map Outputs Channel 1/Data Out 8
//     PlcTask Outputs/GVL_iXlinker.Device_1_EtherCAT.Term_1_EK1200.Term_2_EL6002.COM_RxPDO_Map_Outputs_Channel_1.Data_Out[9] <-> COM RxPDO-Map Outputs Channel 1/Data Out 9
//     PlcTask Outputs/GVL_iXlinker.Device_1_EtherCAT.Term_1_EK1200.Term_2_EL6002.COM_RxPDO_Map_Outputs_Channel_2.Data_Out[0] <-> COM RxPDO-Map Outputs Channel 2/Data Out 0
//     PlcTask Outputs/GVL_iXlinker.Device_1_EtherCAT.Term_1_EK1200.Term_2_EL6002.COM_RxPDO_Map_Outputs_Channel_2.Data_Out[10] <-> COM RxPDO-Map Outputs Channel 2/Data Out 10
//     PlcTask Outputs/GVL_iXlinker.Device_1_EtherCAT.Term_1_EK1200.Term_2_EL6002.COM_RxPDO_Map_Outputs_Channel_2.Data_Out[11] <-> COM RxPDO-Map Outputs Channel 2/Data Out 11
//     PlcTask Outputs/GVL_iXlinker.Device_1_EtherCAT.Term_1_EK1200.Term_2_EL6002.COM_RxPDO_Map_Outputs_Channel_2.Data_Out[12] <-> COM RxPDO-Map Outputs Channel 2/Data Out 12
//     PlcTask Outputs/GVL_iXlinker.Device_1_EtherCAT.Term_1_EK1200.Term_2_EL6002.COM_RxPDO_Map_Outputs_Channel_2.Data_Out[13] <-> COM RxPDO-Map Outputs Channel 2/Data Out 13
//     PlcTask Outputs/GVL_iXlinker.Device_1_EtherCAT.Term_1_EK1200.Term_2_EL6002.COM_RxPDO_Map_Outputs_Channel_2.Data_Out[14] <-> COM RxPDO-Map Outputs Channel 2/Data Out 14
//     PlcTask Outputs/GVL_iXlinker.Device_1_EtherCAT.Term_1_EK1200.Term_2_EL6002.COM_RxPDO_Map_Outputs_Channel_2.Data_Out[15] <-> COM RxPDO-Map Outputs Channel 2/Data Out 15
//     PlcTask Outputs/GVL_iXlinker.Device_1_EtherCAT.Term_1_EK1200.Term_2_EL6002.COM_RxPDO_Map_Outputs_Channel_2.Data_Out[16] <-> COM RxPDO-Map Outputs Channel 2/Data Out 16
//     PlcTask Outputs/GVL_iXlinker.Device_1_EtherCAT.Term_1_EK1200.Term_2_EL6002.COM_RxPDO_Map_Outputs_Channel_2.Data_Out[17] <-> COM RxPDO-Map Outputs Channel 2/Data Out 17
//     PlcTask Outputs/GVL_iXlinker.Device_1_EtherCAT.Term_1_EK1200.Term_2_EL6002.COM_RxPDO_Map_Outputs_Channel_2.Data_Out[18] <-> COM RxPDO-Map Outputs Channel 2/Data Out 18
//     PlcTask Outputs/GVL_iXlinker.Device_1_EtherCAT.Term_1_EK1200.Term_2_EL6002.COM_RxPDO_Map_Outputs_Channel_2.Data_Out[19] <-> COM RxPDO-Map Outputs Channel 2/Data Out 19
//     PlcTask Outputs/GVL_iXlinker.Device_1_EtherCAT.Term_1_EK1200.Term_2_EL6002.COM_RxPDO_Map_Outputs_Channel_2.Data_Out[1] <-> COM RxPDO-Map Outputs Channel 2/Data Out 1
//     PlcTask Outputs/GVL_iXlinker.Device_1_EtherCAT.Term_1_EK1200.Term_2_EL6002.COM_RxPDO_Map_Outputs_Channel_2.Data_Out[20] <-> COM RxPDO-Map Outputs Channel 2/Data Out 20
//     PlcTask Outputs/GVL_iXlinker.Device_1_EtherCAT.Term_1_EK1200.Term_2_EL6002.COM_RxPDO_Map_Outputs_Channel_2.Data_Out[21] <-> COM RxPDO-Map Outputs Channel 2/Data Out 21
//     PlcTask Outputs/GVL_iXlinker.Device_1_EtherCAT.Term_1_EK1200.Term_2_EL6002.COM_RxPDO_Map_Outputs_Channel_2.Data_Out[2] <-> COM RxPDO-Map Outputs Channel 2/Data Out 2
//     PlcTask Outputs/GVL_iXlinker.Device_1_EtherCAT.Term_1_EK1200.Term_2_EL6002.COM_RxPDO_Map_Outputs_Channel_2.Data_Out[3] <-> COM RxPDO-Map Outputs Channel 2/Data Out 3
//     PlcTask Outputs/GVL_iXlinker.Device_1_EtherCAT.Term_1_EK1200.Term_2_EL6002.COM_RxPDO_Map_Outputs_Channel_2.Data_Out[4] <-> COM RxPDO-Map Outputs Channel 2/Data Out 4
//     PlcTask Outputs/GVL_iXlinker.Device_1_EtherCAT.Term_1_EK1200.Term_2_EL6002.COM_RxPDO_Map_Outputs_Channel_2.Data_Out[5] <-> COM RxPDO-Map Outputs Channel 2/Data Out 5
//     PlcTask Outputs/GVL_iXlinker.Device_1_EtherCAT.Term_1_EK1200.Term_2_EL6002.COM_RxPDO_Map_Outputs_Channel_2.Data_Out[6] <-> COM RxPDO-Map Outputs Channel 2/Data Out 6
//     PlcTask Outputs/GVL_iXlinker.Device_1_EtherCAT.Term_1_EK1200.Term_2_EL6002.COM_RxPDO_Map_Outputs_Channel_2.Data_Out[7] <-> COM RxPDO-Map Outputs Channel 2/Data Out 7
//     PlcTask Outputs/GVL_iXlinker.Device_1_EtherCAT.Term_1_EK1200.Term_2_EL6002.COM_RxPDO_Map_Outputs_Channel_2.Data_Out[8] <-> COM RxPDO-Map Outputs Channel 2/Data Out 8
//     PlcTask Outputs/GVL_iXlinker.Device_1_EtherCAT.Term_1_EK1200.Term_2_EL6002.COM_RxPDO_Map_Outputs_Channel_2.Data_Out[9] <-> COM RxPDO-Map Outputs Channel 2/Data Out 9
//   TcoIoTests/TcoIoTests Instance <-> Device 1 (EtherCAT)/Term 1 (EK1200)/Term 3 (EL1809)
//     PlcTask Inputs/GVL_iXlinker.Device_1_EtherCAT.Term_1_EK1200.Term_3_EL1809.Channel_{1..16}.Input <-> Channel {1..16}/Input  (16 links)
//     PlcTask Inputs/GVL_iXlinker.Device_1_EtherCAT.Term_1_EK1200.Term_3_EL1809.InfoData.State <-> InfoData/State
//     PlcTask Inputs/GVL_iXlinker.Device_1_EtherCAT.Term_1_EK1200.Term_3_EL1809.WcState.InputToggle <-> WcState/InputToggle
//     PlcTask Inputs/GVL_iXlinker.Device_1_EtherCAT.Term_1_EK1200.Term_3_EL1809.WcState.WcState <-> WcState/WcState
//   TcoIoTests/TcoIoTests Instance <-> Device 1 (EtherCAT)/Term 1 (EK1200)/Term 4 (EL2809)
//     PlcTask Inputs/GVL_iXlinker.Device_1_EtherCAT.Term_1_EK1200.Term_4_EL2809.InfoData.State <-> InfoData/State
//     PlcTask Inputs/GVL_iXlinker.Device_1_EtherCAT.Term_1_EK1200.Term_4_EL2809.WcState.WcState <-> WcState/WcState
//     PlcTask Outputs/GVL_iXlinker.Device_1_EtherCAT.Term_1_EK1200.Term_4_EL2809.Channel_{1..16}.Output <-> Channel {1..16}/Output  (16 links)
//   TcoIoTests/TcoIoTests Instance <-> Device 1 (EtherCAT)/Term 1 (EK1200)/Term 5 (EL4004)
//     PlcTask Inputs/GVL_iXlinker.Device_1_EtherCAT.Term_1_EK1200.Term_5_EL4004.InfoData.AdsAddr <-> InfoData/AdsAddr
//     PlcTask Inputs/GVL_iXlinker.Device_1_EtherCAT.Term_1_EK1200.Term_5_EL4004.InfoData.State <-> InfoData/State
//     PlcTask Inputs/GVL_iXlinker.Device_1_EtherCAT.Term_1_EK1200.Term_5_EL4004.WcState.WcState <-> WcState/WcState
//     PlcTask Outputs/GVL_iXlinker.Device_1_EtherCAT.Term_1_EK1200.Term_5_EL4004.AO_Outputs_Channel_{1..4}.Analog_output <-> AO Outputs Channel {1..4}/Analog output  (4 links)
//   TcoIoTests/TcoIoTests Instance <-> Device 1 (EtherCAT)/Term 1 (EK1200)/Term 6 (EL2809)
//     PlcTask Inputs/GVL_iXlinker.Device_1_EtherCAT.Term_1_EK1200.Term_6_EL2809.InfoData.State <-> InfoData/State
//     PlcTask Inputs/GVL_iXlinker.Device_1_EtherCAT.Term_1_EK1200.Term_6_EL2809.WcState.WcState <-> WcState/WcState
//     PlcTask Outputs/GVL_iXlinker.Device_1_EtherCAT.Term_1_EK1200.Term_6_EL2809.Channel_{1..16}.Output <-> Channel {1..16}/Output  (16 links)
//   TcoIoTests/TcoIoTests Instance <-> Device 1 (EtherCAT)/Term 1 (EK1200)/Term 7 (EL6001)
//     PlcTask Inputs/GVL_iXlinker.Device_1_EtherCAT.Term_1_EK1200.Term_7_EL6001.COM_Inputs.Data_In[{0..21}] <-> COM Inputs/Data In {0..21}  (22 links)
//     PlcTask Inputs/GVL_iXlinker.Device_1_EtherCAT.Term_1_EK1200.Term_7_EL6001.COM_Inputs.Status/Buffer_full <-> COM Inputs/Status/Buffer full
//     PlcTask Inputs/GVL_iXlinker.Device_1_EtherCAT.Term_1_EK1200.Term_7_EL6001.COM_Inputs.Status/Framing_error <-> COM Inputs/Status/Framing error
//     PlcTask Inputs/GVL_iXlinker.Device_1_EtherCAT.Term_1_EK1200.Term_7_EL6001.COM_Inputs.Status/Init_accepted <-> COM Inputs/Status/Init accepted
//     PlcTask Inputs/GVL_iXlinker.Device_1_EtherCAT.Term_1_EK1200.Term_7_EL6001.COM_Inputs.Status/Input_length <-> COM Inputs/Status/Input length
//     PlcTask Inputs/GVL_iXlinker.Device_1_EtherCAT.Term_1_EK1200.Term_7_EL6001.COM_Inputs.Status/Overrun_error <-> COM Inputs/Status/Overrun error
//     PlcTask Inputs/GVL_iXlinker.Device_1_EtherCAT.Term_1_EK1200.Term_7_EL6001.COM_Inputs.Status/Parity_error <-> COM Inputs/Status/Parity error
//     PlcTask Inputs/GVL_iXlinker.Device_1_EtherCAT.Term_1_EK1200.Term_7_EL6001.COM_Inputs.Status/Receive_request <-> COM Inputs/Status/Receive request
//     PlcTask Inputs/GVL_iXlinker.Device_1_EtherCAT.Term_1_EK1200.Term_7_EL6001.COM_Inputs.Status/Transmit_accepted <-> COM Inputs/Status/Transmit accepted
//     PlcTask Inputs/GVL_iXlinker.Device_1_EtherCAT.Term_1_EK1200.Term_7_EL6001.InfoData.AdsAddr <-> InfoData/AdsAddr
//     PlcTask Inputs/GVL_iXlinker.Device_1_EtherCAT.Term_1_EK1200.Term_7_EL6001.InfoData.State <-> InfoData/State
//     PlcTask Inputs/GVL_iXlinker.Device_1_EtherCAT.Term_1_EK1200.Term_7_EL6001.WcState.InputToggle <-> WcState/InputToggle
//     PlcTask Inputs/GVL_iXlinker.Device_1_EtherCAT.Term_1_EK1200.Term_7_EL6001.WcState.WcState <-> WcState/WcState
//     PlcTask Outputs/GVL_iXlinker.Device_1_EtherCAT.Term_1_EK1200.Term_7_EL6001.COM_Outputs.Ctrl/Init_request <-> COM Outputs/Ctrl/Init request
//     PlcTask Outputs/GVL_iXlinker.Device_1_EtherCAT.Term_1_EK1200.Term_7_EL6001.COM_Outputs.Ctrl/Output_length <-> COM Outputs/Ctrl/Output length
//     PlcTask Outputs/GVL_iXlinker.Device_1_EtherCAT.Term_1_EK1200.Term_7_EL6001.COM_Outputs.Ctrl/Receive_accepted <-> COM Outputs/Ctrl/Receive accepted
//     PlcTask Outputs/GVL_iXlinker.Device_1_EtherCAT.Term_1_EK1200.Term_7_EL6001.COM_Outputs.Ctrl/Send_continues <-> COM Outputs/Ctrl/Send continues
//     PlcTask Outputs/GVL_iXlinker.Device_1_EtherCAT.Term_1_EK1200.Term_7_EL6001.COM_Outputs.Ctrl/Transmit_request <-> COM Outputs/Ctrl/Transmit request
//     PlcTask Outputs/GVL_iXlinker.Device_1_EtherCAT.Term_1_EK1200.Term_7_EL6001.COM_Outputs.Data_Out[{0..21}] <-> COM Outputs/Data Out {0..21}  (22 links)
//   TcoIoTests/TcoIoTests Instance <-> Device 4 (EtherCAT)
//     PlcTask Inputs/GVL_iXlinker.Device_4_EtherCAT.InfoData.AmsNetId <-> InfoData/AmsNetId
//     PlcTask Inputs/GVL_iXlinker.Device_4_EtherCAT.InfoData.CfgSlaveCount <-> InfoData/CfgSlaveCount
//     PlcTask Inputs/GVL_iXlinker.Device_4_EtherCAT.InfoData.ChangeCount <-> InfoData/ChangeCount
//     PlcTask Inputs/GVL_iXlinker.Device_4_EtherCAT.InfoData.DevId <-> InfoData/DevId
//     PlcTask Inputs/GVL_iXlinker.Device_4_EtherCAT.Inputs.DevState <-> Inputs/DevState
//     PlcTask Inputs/GVL_iXlinker.Device_4_EtherCAT.Inputs.Frm0InputToggle <-> Inputs/Frm0InputToggle
//     PlcTask Inputs/GVL_iXlinker.Device_4_EtherCAT.Inputs.Frm0State <-> Inputs/Frm0State
//     PlcTask Inputs/GVL_iXlinker.Device_4_EtherCAT.Inputs.Frm0WcState <-> Inputs/Frm0WcState
//     PlcTask Inputs/GVL_iXlinker.Device_4_EtherCAT.Inputs.SlaveCount <-> Inputs/SlaveCount
//     PlcTask Outputs/GVL_iXlinker.Device_4_EtherCAT.Outputs.DevCtrl <-> Outputs/DevCtrl
//     PlcTask Outputs/GVL_iXlinker.Device_4_EtherCAT.Outputs.Frm0Ctrl <-> Outputs/Frm0Ctrl
//     PlcTask Outputs/GVL_iXlinker.Device_4_EtherCAT.Outputs.Frm0WcCtrl <-> Outputs/Frm0WcCtrl
//   TcoIoTests/TcoIoTests Instance <-> Device 4 (EtherCAT)/Term 9 (EK1100)
//     PlcTask Inputs/GVL_iXlinker.Device_4_EtherCAT.Term_9_EK1100.InfoData.State <-> InfoData/State

CONFIGURATION TcoIoTests
    RESOURCE PLC ON TwinCAT3
        TASK PlcTask(INTERVAL := T#15ms, PRIORITY := 6);
        PROGRAM MAIN WITH PlcTask : MAIN;
    END_RESOURCE
END_CONFIGURATION

// ---- DUTs/IO/PdoEntries/Status_3D84275F.TcDUT
{attribute 'GeneratedUsingTerminal: EL6002-0000-0019'}
{attribute addProperty BoxType "EL6002-0000-0019"}
{attribute addProperty Id "Transmit_acceptedBOOL1Receive_requestBOOL1Init_acceptedBOOL1Buffer_fullBOOL1Parity_errorBOOL1Framing_errorBOOL1Overrun_errorBOOL1Input_lengthUSINT1"}
{attribute addProperty CRC "1032071007"}
{attribute addProperty Size "8"}
TYPE Status_3D84275F :
STRUCT
    {attribute addProperty Name "Transmit_accepted"}
    Transmit_accepted : BOOL;
    {attribute addProperty Name "Receive_request"}
    Receive_request : BOOL;
    {attribute addProperty Name "Init_accepted"}
    Init_accepted : BOOL;
    {attribute addProperty Name "Buffer_full"}
    Buffer_full : BOOL;
    {attribute addProperty Name "Parity_error"}
    Parity_error : BOOL;
    {attribute addProperty Name "Framing_error"}
    Framing_error : BOOL;
    {attribute addProperty Name "Overrun_error"}
    Overrun_error : BOOL;
    {attribute addProperty Name "Input_length"}
    Input_length : USINT;
END_STRUCT
END_TYPE

// ---- DUTs/IO/PdoEntries/Ctrl_1EFB4D3B.TcDUT
{attribute 'GeneratedUsingTerminal: EL6002-0000-0019'}
{attribute addProperty BoxType "EL6002-0000-0019"}
{attribute addProperty Id "Transmit_requestBOOL1Receive_acceptedBOOL1Init_requestBOOL1Send_continuousBOOL1Output_lengthUSINT1"}
{attribute addProperty CRC "519785787"}
{attribute addProperty Size "5"}
TYPE Ctrl_1EFB4D3B :
STRUCT
    {attribute addProperty Name "Transmit_request"}
    Transmit_request : BOOL;
    {attribute addProperty Name "Receive_accepted"}
    Receive_accepted : BOOL;
    {attribute addProperty Name "Init_request"}
    Init_request : BOOL;
    {attribute addProperty Name "Send_continuous"}
    Send_continuous : BOOL;
    {attribute addProperty Name "Output_length"}
    Output_length : USINT;
END_STRUCT
END_TYPE

// ---- DUTs/IO/PdoEntries/Ctrl_71604E86.TcDUT
{attribute 'GeneratedUsingTerminal: EL6001-0000-0020'}
{attribute addProperty BoxType "EL6001-0000-0020"}
{attribute addProperty Id "Transmit_requestBOOL1Receive_acceptedBOOL1Init_requestBOOL1Send_continuesBOOL1Output_lengthUSINT1"}
{attribute addProperty CRC "1902136966"}
{attribute addProperty Size "5"}
TYPE Ctrl_71604E86 :
STRUCT
    {attribute addProperty Name "Transmit_request"}
    Transmit_request : BOOL;
    {attribute addProperty Name "Receive_accepted"}
    Receive_accepted : BOOL;
    {attribute addProperty Name "Init_request"}
    Init_request : BOOL;
    {attribute addProperty Name "Send_continues"}
    Send_continues : BOOL;
    {attribute addProperty Name "Output_length"}
    Output_length : USINT;
END_STRUCT
END_TYPE

// ---- DUTs/IO/PdoEntries/Status_B0753356.TcDUT
{attribute 'GeneratedUsingTerminal: EL3174-0002-0017'}
{attribute addProperty BoxType "EL3174-0002-0017"}
{attribute addProperty Id "UnderrangeBOOL1OverrangeBOOL1Limit_1BYTE1Limit_2BYTE1ErrorBOOL1Sync_errorBOOL1TxPDO_StateBOOL1TxPDO_ToggleBOOL1"}
{attribute addProperty CRC "2960470870"}
{attribute addProperty Size "8"}
TYPE Status_B0753356 :
STRUCT
    {attribute addProperty Name "Underrange"}
    Underrange : BOOL;
    {attribute addProperty Name "Overrange"}
    Overrange : BOOL;
    {attribute addProperty Name "Limit_1"}
    Limit_1 : BYTE;
    {attribute addProperty Name "Limit_2"}
    Limit_2 : BYTE;
    {attribute addProperty Name "Error"}
    Error : BOOL;
    {attribute addProperty Name "Sync_error"}
    Sync_error : BOOL;
    {attribute addProperty Name "TxPDO_State"}
    TxPDO_State : BOOL;
    {attribute addProperty Name "TxPDO_Toggle"}
    TxPDO_Toggle : BOOL;
END_STRUCT
END_TYPE

// ---- DUTs/IO/PdoEntries/Status_F2CE6D91.TcDUT
{attribute 'GeneratedUsingTerminal: EL3011-0000-0018'}
{attribute addProperty BoxType "EL3011-0000-0018"}
{attribute addProperty Id "UnderrangeBOOL1OverrangeBOOL1Limit_1BYTE1Limit_2BYTE1ErrorBOOL1TxPDO_StateBOOL1TxPDO_ToggleBOOL1"}
{attribute addProperty CRC "4073614737"}
{attribute addProperty Size "7"}
TYPE Status_F2CE6D91 :
STRUCT
    {attribute addProperty Name "Underrange"}
    Underrange : BOOL;
    {attribute addProperty Name "Overrange"}
    Overrange : BOOL;
    {attribute addProperty Name "Limit_1"}
    Limit_1 : BYTE;
    {attribute addProperty Name "Limit_2"}
    Limit_2 : BYTE;
    {attribute addProperty Name "Error"}
    Error : BOOL;
    {attribute addProperty Name "TxPDO_State"}
    TxPDO_State : BOOL;
    {attribute addProperty Name "TxPDO_Toggle"}
    TxPDO_Toggle : BOOL;
END_STRUCT
END_TYPE

// ---- DUTs/IO/PdoEntries/U1_Status_DC903920.TcDUT
{attribute 'GeneratedUsingTerminal: EL3773-0000-0021'}
{attribute addProperty BoxType "EL3773-0000-0021"}
{attribute addProperty Id "UnderrangeBOOL1OverrangeBOOL1Limit_xBYTE1ErrorBOOL1Sync_errorBOOL1TxPDO_StateBOOL1TxPDO_ToggleBOOL1"}
{attribute addProperty CRC "3700439328"}
{attribute addProperty Size "7"}
TYPE U1_Status_DC903920 :
STRUCT
    {attribute addProperty Name "Underrange"}
    Underrange : BOOL;
    {attribute addProperty Name "Overrange"}
    Overrange : BOOL;
    {attribute addProperty Name "Limit_x"}
    Limit_x : BYTE;
    {attribute addProperty Name "Error"}
    Error : BOOL;
    {attribute addProperty Name "Sync_error"}
    Sync_error : BOOL;
    {attribute addProperty Name "TxPDO_State"}
    TxPDO_State : BOOL;
    {attribute addProperty Name "TxPDO_Toggle"}
    TxPDO_Toggle : BOOL;
END_STRUCT
END_TYPE

// ---- DUTs/IO/PdoEntries/U1_Samples_25492287.TcDUT
{attribute 'GeneratedUsingTerminal: EL3773-0000-0021'}
{attribute addProperty BoxType "EL3773-0000-0021"}
{attribute addProperty Id "ARRAY_0INT2ARRAY_1INT2ARRAY_2INT2ARRAY_3INT2ARRAY_4INT2ARRAY_5INT2ARRAY_6INT2ARRAY_7INT2ARRAY_8INT2ARRAY_9INT2"}
{attribute addProperty CRC "625549959"}
{attribute addProperty Size "20"}
TYPE U1_Samples_25492287 :
STRUCT
    {attribute addProperty Name "ARRAY_0"}
    ARRAY_0 : INT;
    {attribute addProperty Name "ARRAY_1"}
    ARRAY_1 : INT;
    {attribute addProperty Name "ARRAY_2"}
    ARRAY_2 : INT;
    {attribute addProperty Name "ARRAY_3"}
    ARRAY_3 : INT;
    {attribute addProperty Name "ARRAY_4"}
    ARRAY_4 : INT;
    {attribute addProperty Name "ARRAY_5"}
    ARRAY_5 : INT;
    {attribute addProperty Name "ARRAY_6"}
    ARRAY_6 : INT;
    {attribute addProperty Name "ARRAY_7"}
    ARRAY_7 : INT;
    {attribute addProperty Name "ARRAY_8"}
    ARRAY_8 : INT;
    {attribute addProperty Name "ARRAY_9"}
    ARRAY_9 : INT;
END_STRUCT
END_TYPE

// ---- DUTs/IO/PdoEntries/I1_Status_DC903920.TcDUT
{attribute 'GeneratedUsingTerminal: EL3773-0000-0021'}
{attribute addProperty BoxType "EL3773-0000-0021"}
{attribute addProperty Id "UnderrangeBOOL1OverrangeBOOL1Limit_xBYTE1ErrorBOOL1Sync_errorBOOL1TxPDO_StateBOOL1TxPDO_ToggleBOOL1"}
{attribute addProperty CRC "3700439328"}
{attribute addProperty Size "7"}
TYPE I1_Status_DC903920 :
STRUCT
    {attribute addProperty Name "Underrange"}
    Underrange : BOOL;
    {attribute addProperty Name "Overrange"}
    Overrange : BOOL;
    {attribute addProperty Name "Limit_x"}
    Limit_x : BYTE;
    {attribute addProperty Name "Error"}
    Error : BOOL;
    {attribute addProperty Name "Sync_error"}
    Sync_error : BOOL;
    {attribute addProperty Name "TxPDO_State"}
    TxPDO_State : BOOL;
    {attribute addProperty Name "TxPDO_Toggle"}
    TxPDO_Toggle : BOOL;
END_STRUCT
END_TYPE

// ---- DUTs/IO/PdoEntries/I1_Samples_25492287.TcDUT
{attribute 'GeneratedUsingTerminal: EL3773-0000-0021'}
{attribute addProperty BoxType "EL3773-0000-0021"}
{attribute addProperty Id "ARRAY_0INT2ARRAY_1INT2ARRAY_2INT2ARRAY_3INT2ARRAY_4INT2ARRAY_5INT2ARRAY_6INT2ARRAY_7INT2ARRAY_8INT2ARRAY_9INT2"}
{attribute addProperty CRC "625549959"}
{attribute addProperty Size "20"}
TYPE I1_Samples_25492287 :
STRUCT
    {attribute addProperty Name "ARRAY_0"}
    ARRAY_0 : INT;
    {attribute addProperty Name "ARRAY_1"}
    ARRAY_1 : INT;
    {attribute addProperty Name "ARRAY_2"}
    ARRAY_2 : INT;
    {attribute addProperty Name "ARRAY_3"}
    ARRAY_3 : INT;
    {attribute addProperty Name "ARRAY_4"}
    ARRAY_4 : INT;
    {attribute addProperty Name "ARRAY_5"}
    ARRAY_5 : INT;
    {attribute addProperty Name "ARRAY_6"}
    ARRAY_6 : INT;
    {attribute addProperty Name "ARRAY_7"}
    ARRAY_7 : INT;
    {attribute addProperty Name "ARRAY_8"}
    ARRAY_8 : INT;
    {attribute addProperty Name "ARRAY_9"}
    ARRAY_9 : INT;
END_STRUCT
END_TYPE

// ---- DUTs/IO/PdoEntries/U2_Status_DC903920.TcDUT
{attribute 'GeneratedUsingTerminal: EL3773-0000-0021'}
{attribute addProperty BoxType "EL3773-0000-0021"}
{attribute addProperty Id "UnderrangeBOOL1OverrangeBOOL1Limit_xBYTE1ErrorBOOL1Sync_errorBOOL1TxPDO_StateBOOL1TxPDO_ToggleBOOL1"}
{attribute addProperty CRC "3700439328"}
{attribute addProperty Size "7"}
TYPE U2_Status_DC903920 :
STRUCT
    {attribute addProperty Name "Underrange"}
    Underrange : BOOL;
    {attribute addProperty Name "Overrange"}
    Overrange : BOOL;
    {attribute addProperty Name "Limit_x"}
    Limit_x : BYTE;
    {attribute addProperty Name "Error"}
    Error : BOOL;
    {attribute addProperty Name "Sync_error"}
    Sync_error : BOOL;
    {attribute addProperty Name "TxPDO_State"}
    TxPDO_State : BOOL;
    {attribute addProperty Name "TxPDO_Toggle"}
    TxPDO_Toggle : BOOL;
END_STRUCT
END_TYPE

// ---- DUTs/IO/PdoEntries/U2_Samples_25492287.TcDUT
{attribute 'GeneratedUsingTerminal: EL3773-0000-0021'}
{attribute addProperty BoxType "EL3773-0000-0021"}
{attribute addProperty Id "ARRAY_0INT2ARRAY_1INT2ARRAY_2INT2ARRAY_3INT2ARRAY_4INT2ARRAY_5INT2ARRAY_6INT2ARRAY_7INT2ARRAY_8INT2ARRAY_9INT2"}
{attribute addProperty CRC "625549959"}
{attribute addProperty Size "20"}
TYPE U2_Samples_25492287 :
STRUCT
    {attribute addProperty Name "ARRAY_0"}
    ARRAY_0 : INT;
    {attribute addProperty Name "ARRAY_1"}
    ARRAY_1 : INT;
    {attribute addProperty Name "ARRAY_2"}
    ARRAY_2 : INT;
    {attribute addProperty Name "ARRAY_3"}
    ARRAY_3 : INT;
    {attribute addProperty Name "ARRAY_4"}
    ARRAY_4 : INT;
    {attribute addProperty Name "ARRAY_5"}
    ARRAY_5 : INT;
    {attribute addProperty Name "ARRAY_6"}
    ARRAY_6 : INT;
    {attribute addProperty Name "ARRAY_7"}
    ARRAY_7 : INT;
    {attribute addProperty Name "ARRAY_8"}
    ARRAY_8 : INT;
    {attribute addProperty Name "ARRAY_9"}
    ARRAY_9 : INT;
END_STRUCT
END_TYPE

// ---- DUTs/IO/PdoEntries/I2_Status_DC903920.TcDUT
{attribute 'GeneratedUsingTerminal: EL3773-0000-0021'}
{attribute addProperty BoxType "EL3773-0000-0021"}
{attribute addProperty Id "UnderrangeBOOL1OverrangeBOOL1Limit_xBYTE1ErrorBOOL1Sync_errorBOOL1TxPDO_StateBOOL1TxPDO_ToggleBOOL1"}
{attribute addProperty CRC "3700439328"}
{attribute addProperty Size "7"}
TYPE I2_Status_DC903920 :
STRUCT
    {attribute addProperty Name "Underrange"}
    Underrange : BOOL;
    {attribute addProperty Name "Overrange"}
    Overrange : BOOL;
    {attribute addProperty Name "Limit_x"}
    Limit_x : BYTE;
    {attribute addProperty Name "Error"}
    Error : BOOL;
    {attribute addProperty Name "Sync_error"}
    Sync_error : BOOL;
    {attribute addProperty Name "TxPDO_State"}
    TxPDO_State : BOOL;
    {attribute addProperty Name "TxPDO_Toggle"}
    TxPDO_Toggle : BOOL;
END_STRUCT
END_TYPE

// ---- DUTs/IO/PdoEntries/I2_Samples_25492287.TcDUT
{attribute 'GeneratedUsingTerminal: EL3773-0000-0021'}
{attribute addProperty BoxType "EL3773-0000-0021"}
{attribute addProperty Id "ARRAY_0INT2ARRAY_1INT2ARRAY_2INT2ARRAY_3INT2ARRAY_4INT2ARRAY_5INT2ARRAY_6INT2ARRAY_7INT2ARRAY_8INT2ARRAY_9INT2"}
{attribute addProperty CRC "625549959"}
{attribute addProperty Size "20"}
TYPE I2_Samples_25492287 :
STRUCT
    {attribute addProperty Name "ARRAY_0"}
    ARRAY_0 : INT;
    {attribute addProperty Name "ARRAY_1"}
    ARRAY_1 : INT;
    {attribute addProperty Name "ARRAY_2"}
    ARRAY_2 : INT;
    {attribute addProperty Name "ARRAY_3"}
    ARRAY_3 : INT;
    {attribute addProperty Name "ARRAY_4"}
    ARRAY_4 : INT;
    {attribute addProperty Name "ARRAY_5"}
    ARRAY_5 : INT;
    {attribute addProperty Name "ARRAY_6"}
    ARRAY_6 : INT;
    {attribute addProperty Name "ARRAY_7"}
    ARRAY_7 : INT;
    {attribute addProperty Name "ARRAY_8"}
    ARRAY_8 : INT;
    {attribute addProperty Name "ARRAY_9"}
    ARRAY_9 : INT;
END_STRUCT
END_TYPE

// ---- DUTs/IO/PdoEntries/U3_Status_DC903920.TcDUT
{attribute 'GeneratedUsingTerminal: EL3773-0000-0021'}
{attribute addProperty BoxType "EL3773-0000-0021"}
{attribute addProperty Id "UnderrangeBOOL1OverrangeBOOL1Limit_xBYTE1ErrorBOOL1Sync_errorBOOL1TxPDO_StateBOOL1TxPDO_ToggleBOOL1"}
{attribute addProperty CRC "3700439328"}
{attribute addProperty Size "7"}
TYPE U3_Status_DC903920 :
STRUCT
    {attribute addProperty Name "Underrange"}
    Underrange : BOOL;
    {attribute addProperty Name "Overrange"}
    Overrange : BOOL;
    {attribute addProperty Name "Limit_x"}
    Limit_x : BYTE;
    {attribute addProperty Name "Error"}
    Error : BOOL;
    {attribute addProperty Name "Sync_error"}
    Sync_error : BOOL;
    {attribute addProperty Name "TxPDO_State"}
    TxPDO_State : BOOL;
    {attribute addProperty Name "TxPDO_Toggle"}
    TxPDO_Toggle : BOOL;
END_STRUCT
END_TYPE

// ---- DUTs/IO/PdoEntries/U3_Samples_25492287.TcDUT
{attribute 'GeneratedUsingTerminal: EL3773-0000-0021'}
{attribute addProperty BoxType "EL3773-0000-0021"}
{attribute addProperty Id "ARRAY_0INT2ARRAY_1INT2ARRAY_2INT2ARRAY_3INT2ARRAY_4INT2ARRAY_5INT2ARRAY_6INT2ARRAY_7INT2ARRAY_8INT2ARRAY_9INT2"}
{attribute addProperty CRC "625549959"}
{attribute addProperty Size "20"}
TYPE U3_Samples_25492287 :
STRUCT
    {attribute addProperty Name "ARRAY_0"}
    ARRAY_0 : INT;
    {attribute addProperty Name "ARRAY_1"}
    ARRAY_1 : INT;
    {attribute addProperty Name "ARRAY_2"}
    ARRAY_2 : INT;
    {attribute addProperty Name "ARRAY_3"}
    ARRAY_3 : INT;
    {attribute addProperty Name "ARRAY_4"}
    ARRAY_4 : INT;
    {attribute addProperty Name "ARRAY_5"}
    ARRAY_5 : INT;
    {attribute addProperty Name "ARRAY_6"}
    ARRAY_6 : INT;
    {attribute addProperty Name "ARRAY_7"}
    ARRAY_7 : INT;
    {attribute addProperty Name "ARRAY_8"}
    ARRAY_8 : INT;
    {attribute addProperty Name "ARRAY_9"}
    ARRAY_9 : INT;
END_STRUCT
END_TYPE

// ---- DUTs/IO/PdoEntries/I3_Status_DC903920.TcDUT
{attribute 'GeneratedUsingTerminal: EL3773-0000-0021'}
{attribute addProperty BoxType "EL3773-0000-0021"}
{attribute addProperty Id "UnderrangeBOOL1OverrangeBOOL1Limit_xBYTE1ErrorBOOL1Sync_errorBOOL1TxPDO_StateBOOL1TxPDO_ToggleBOOL1"}
{attribute addProperty CRC "3700439328"}
{attribute addProperty Size "7"}
TYPE I3_Status_DC903920 :
STRUCT
    {attribute addProperty Name "Underrange"}
    Underrange : BOOL;
    {attribute addProperty Name "Overrange"}
    Overrange : BOOL;
    {attribute addProperty Name "Limit_x"}
    Limit_x : BYTE;
    {attribute addProperty Name "Error"}
    Error : BOOL;
    {attribute addProperty Name "Sync_error"}
    Sync_error : BOOL;
    {attribute addProperty Name "TxPDO_State"}
    TxPDO_State : BOOL;
    {attribute addProperty Name "TxPDO_Toggle"}
    TxPDO_Toggle : BOOL;
END_STRUCT
END_TYPE

// ---- DUTs/IO/PdoEntries/I3_Samples_25492287.TcDUT
{attribute 'GeneratedUsingTerminal: EL3773-0000-0021'}
{attribute addProperty BoxType "EL3773-0000-0021"}
{attribute addProperty Id "ARRAY_0INT2ARRAY_1INT2ARRAY_2INT2ARRAY_3INT2ARRAY_4INT2ARRAY_5INT2ARRAY_6INT2ARRAY_7INT2ARRAY_8INT2ARRAY_9INT2"}
{attribute addProperty CRC "625549959"}
{attribute addProperty Size "20"}
TYPE I3_Samples_25492287 :
STRUCT
    {attribute addProperty Name "ARRAY_0"}
    ARRAY_0 : INT;
    {attribute addProperty Name "ARRAY_1"}
    ARRAY_1 : INT;
    {attribute addProperty Name "ARRAY_2"}
    ARRAY_2 : INT;
    {attribute addProperty Name "ARRAY_3"}
    ARRAY_3 : INT;
    {attribute addProperty Name "ARRAY_4"}
    ARRAY_4 : INT;
    {attribute addProperty Name "ARRAY_5"}
    ARRAY_5 : INT;
    {attribute addProperty Name "ARRAY_6"}
    ARRAY_6 : INT;
    {attribute addProperty Name "ARRAY_7"}
    ARRAY_7 : INT;
    {attribute addProperty Name "ARRAY_8"}
    ARRAY_8 : INT;
    {attribute addProperty Name "ARRAY_9"}
    ARRAY_9 : INT;
END_STRUCT
END_TYPE

// ---- DUTs/IO/PdoEntries/StartTimeNextLatch_02E0C1C8.TcDUT
{attribute 'GeneratedUsingTerminal: EL3773-0000-0021'}
{attribute addProperty BoxType "EL3773-0000-0021"}
{attribute addProperty Id "LowUDINT4HiUDINT4"}
{attribute addProperty CRC "48284104"}
{attribute addProperty Size "8"}
TYPE StartTimeNextLatch_02E0C1C8 :
STRUCT
    {attribute addProperty Name "Low"}
    Low : UDINT;
    {attribute addProperty Name "Hi"}
    Hi : UDINT;
END_STRUCT
END_TYPE

// ---- DUTs/IO/PdoEntries/Status_642C2ED1.TcDUT
{attribute 'GeneratedUsingTerminal: EL2258-0000-0017'}
{attribute addProperty BoxType "EL2258-0000-0017"}
{attribute addProperty Id "Output_short_circuitBOOL1Output_buffer_overflowBOOL1Output_stateBOOL1Input_cycle_counterBYTE1Output_order_feedbackUSINT1Events_in_output_bufferUSINT1"}
{attribute addProperty CRC "1680617169"}
{attribute addProperty Size "6"}
TYPE Status_642C2ED1 :
STRUCT
    {attribute addProperty Name "Output_short_circuit"}
    Output_short_circuit : BOOL;
    {attribute addProperty Name "Output_buffer_overflow"}
    Output_buffer_overflow : BOOL;
    {attribute addProperty Name "Output_state"}
    Output_state : BOOL;
    {attribute addProperty Name "Input_cycle_counter"}
    Input_cycle_counter : BYTE;
    {attribute addProperty Name "Output_order_feedback"}
    Output_order_feedback : USINT;
    {attribute addProperty Name "Events_in_output_buffer"}
    Events_in_output_buffer : USINT;
END_STRUCT
END_TYPE

// ---- DUTs/IO/PdoEntries/Ctrl_77460BD3.TcDUT
{attribute 'GeneratedUsingTerminal: EL2258-0000-0017'}
{attribute addProperty BoxType "EL2258-0000-0017"}
{attribute addProperty Id "Output_buffer_resetBOOL1Manual_output_stateBOOL1Force_orderBOOL1Enable_manual_operationBOOL1Output_order_counterUSINT1No_of_output_eventsUSINT1"}
{attribute addProperty CRC "2001079251"}
{attribute addProperty Size "6"}
TYPE Ctrl_77460BD3 :
STRUCT
    {attribute addProperty Name "Output_buffer_reset"}
    Output_buffer_reset : BOOL;
    {attribute addProperty Name "Manual_output_state"}
    Manual_output_state : BOOL;
    {attribute addProperty Name "Force_order"}
    Force_order : BOOL;
    {attribute addProperty Name "Enable_manual_operation"}
    Enable_manual_operation : BOOL;
    {attribute addProperty Name "Output_order_counter"}
    Output_order_counter : USINT;
    {attribute addProperty Name "No_of_output_events"}
    No_of_output_events : USINT;
END_STRUCT
END_TYPE

// ---- DUTs/IO/PdoEntries/Outputs_A910484D.TcDUT
{attribute 'GeneratedUsingTerminal: EL2258-0000-0017'}
{attribute addProperty BoxType "EL2258-0000-0017"}
{attribute addProperty Id "Output_event_state_1BOOL1Output_event_state_2BOOL1Output_event_state_3BOOL1Output_event_state_4BOOL1Output_event_state_5BOOL1Output_event_state_6BOOL1Output_event_state_7BOOL1Output_event_state_8BOOL1Output_event_state_9BOOL1Output_event_state_10BOOL1"}
{attribute addProperty CRC "2836416589"}
{attribute addProperty Size "10"}
TYPE Outputs_A910484D :
STRUCT
    {attribute addProperty Name "Output_event_state_1"}
    Output_event_state_1 : BOOL;
    {attribute addProperty Name "Output_event_state_2"}
    Output_event_state_2 : BOOL;
    {attribute addProperty Name "Output_event_state_3"}
    Output_event_state_3 : BOOL;
    {attribute addProperty Name "Output_event_state_4"}
    Output_event_state_4 : BOOL;
    {attribute addProperty Name "Output_event_state_5"}
    Output_event_state_5 : BOOL;
    {attribute addProperty Name "Output_event_state_6"}
    Output_event_state_6 : BOOL;
    {attribute addProperty Name "Output_event_state_7"}
    Output_event_state_7 : BOOL;
    {attribute addProperty Name "Output_event_state_8"}
    Output_event_state_8 : BOOL;
    {attribute addProperty Name "Output_event_state_9"}
    Output_event_state_9 : BOOL;
    {attribute addProperty Name "Output_event_state_10"}
    Output_event_state_10 : BOOL;
END_STRUCT
END_TYPE

// ---- DUTs/IO/PdoEntries/Status_B6795845.TcDUT
{attribute 'GeneratedUsingTerminal: EL7332-0000-0024'}
{attribute addProperty BoxType "EL7332-0000-0024"}
{attribute addProperty Id "Ready_to_enableBOOL1ReadyBOOL1WarningBOOL1ErrorBOOL1Moving_positiveBOOL1Moving_negativeBOOL1Torque_reducedBOOL1Digital_input_1BOOL1Digital_input_2BOOL1Sync_errorBOOL1TxPDO_ToggleBOOL1"}
{attribute addProperty CRC "3061405765"}
{attribute addProperty Size "11"}
TYPE Status_B6795845 :
STRUCT
    {attribute addProperty Name "Ready_to_enable"}
    Ready_to_enable : BOOL;
    {attribute addProperty Name "Ready"}
    Ready : BOOL;
    {attribute addProperty Name "Warning"}
    Warning : BOOL;
    {attribute addProperty Name "Error"}
    Error : BOOL;
    {attribute addProperty Name "Moving_positive"}
    Moving_positive : BOOL;
    {attribute addProperty Name "Moving_negative"}
    Moving_negative : BOOL;
    {attribute addProperty Name "Torque_reduced"}
    Torque_reduced : BOOL;
    {attribute addProperty Name "Digital_input_1"}
    Digital_input_1 : BOOL;
    {attribute addProperty Name "Digital_input_2"}
    Digital_input_2 : BOOL;
    {attribute addProperty Name "Sync_error"}
    Sync_error : BOOL;
    {attribute addProperty Name "TxPDO_Toggle"}
    TxPDO_Toggle : BOOL;
END_STRUCT
END_TYPE

// ---- DUTs/IO/PdoEntries/Control_C948E0F2.TcDUT
{attribute 'GeneratedUsingTerminal: EL7332-0000-0024'}
{attribute addProperty BoxType "EL7332-0000-0024"}
{attribute addProperty Id "EnableBOOL1ResetBOOL1Reduce_torqueBOOL1"}
{attribute addProperty CRC "3376996594"}
{attribute addProperty Size "3"}
TYPE Control_C948E0F2 :
STRUCT
    {attribute addProperty Name "Enable"}
    Enable : BOOL;
    {attribute addProperty Name "Reset"}
    Reset : BOOL;
    {attribute addProperty Name "Reduce_torque"}
    Reduce_torque : BOOL;
END_STRUCT
END_TYPE

// ---- DUTs/IO/PdoEntries/Status_439F40C3.TcDUT
{attribute 'GeneratedUsingTerminal: EL3692-0000-0020'}
{attribute addProperty BoxType "EL3692-0000-0020"}
{attribute addProperty Id "UnderrangeBOOL1OverrangeBOOL1Extended_rangeBOOL1Data_invalidBOOL1Range_invalidBOOL1Autorange_disabledBOOL1ErrorBOOL1Steady_stateBOOL1TxPDO_StateBOOL1TxPDO_ToggleBOOL1"}
{attribute addProperty CRC "1134510275"}
{attribute addProperty Size "10"}
TYPE Status_439F40C3 :
STRUCT
    {attribute addProperty Name "Underrange"}
    Underrange : BOOL;
    {attribute addProperty Name "Overrange"}
    Overrange : BOOL;
    {attribute addProperty Name "Extended_range"}
    Extended_range : BOOL;
    {attribute addProperty Name "Data_invalid"}
    Data_invalid : BOOL;
    {attribute addProperty Name "Range_invalid"}
    Range_invalid : BOOL;
    {attribute addProperty Name "Autorange_disabled"}
    Autorange_disabled : BOOL;
    {attribute addProperty Name "Error"}
    Error : BOOL;
    {attribute addProperty Name "Steady_state"}
    Steady_state : BOOL;
    {attribute addProperty Name "TxPDO_State"}
    TxPDO_State : BOOL;
    {attribute addProperty Name "TxPDO_Toggle"}
    TxPDO_Toggle : BOOL;
END_STRUCT
END_TYPE

// ---- DUTs/IO/PdoEntries/Settings_24C04940.TcDUT
{attribute 'GeneratedUsingTerminal: EL3692-0000-0020'}
{attribute addProperty BoxType "EL3692-0000-0020"}
{attribute addProperty Id "ModeBYTE1RangeSINT1"}
{attribute addProperty CRC "616581440"}
{attribute addProperty Size "2"}
TYPE Settings_24C04940 :
STRUCT
    {attribute addProperty Name "Mode"}
    Mode : BYTE;
    {attribute addProperty Name "Range"}
    Range : SINT;
END_STRUCT
END_TYPE

// ---- DUTs/IO/PdoEntries/Control_E49DBA1B.TcDUT
{attribute 'GeneratedUsingTerminal: EL3692-0000-0020'}
{attribute addProperty BoxType "EL3692-0000-0020"}
{attribute addProperty Id "Disable_autorangeBOOL1Start_conversionBOOL1ModeBYTE1RangeSINT1"}
{attribute addProperty CRC "3835542043"}
{attribute addProperty Size "4"}
TYPE Control_E49DBA1B :
STRUCT
    {attribute addProperty Name "Disable_autorange"}
    Disable_autorange : BOOL;
    {attribute addProperty Name "Start_conversion"}
    Start_conversion : BOOL;
    {attribute addProperty Name "Mode"}
    Mode : BYTE;
    {attribute addProperty Name "Range"}
    Range : SINT;
END_STRUCT
END_TYPE

// ---- DUTs/IO/PdoEntries/Status_8CBE219F.TcDUT
{attribute 'GeneratedUsingTerminal: EL7041-1000-0021'}
{attribute addProperty BoxType "EL7041-1000-0021"}
{attribute addProperty Id "Latch_C_validBOOL1Latch_extern_validBOOL1Set_counter_doneBOOL1Counter_underflowBOOL1Counter_overflowBOOL1Extrapolation_stallBOOL1Status_of_input_ABOOL1Status_of_input_BBOOL1Status_of_input_CBOOL1Status_of_extern_latchBOOL1Sync_errorBOOL1TxPDO_ToggleBOOL1"}
{attribute addProperty CRC "2361270687"}
{attribute addProperty Size "12"}
TYPE Status_8CBE219F :
STRUCT
    {attribute addProperty Name "Latch_C_valid"}
    Latch_C_valid : BOOL;
    {attribute addProperty Name "Latch_extern_valid"}
    Latch_extern_valid : BOOL;
    {attribute addProperty Name "Set_counter_done"}
    Set_counter_done : BOOL;
    {attribute addProperty Name "Counter_underflow"}
    Counter_underflow : BOOL;
    {attribute addProperty Name "Counter_overflow"}
    Counter_overflow : BOOL;
    {attribute addProperty Name "Extrapolation_stall"}
    Extrapolation_stall : BOOL;
    {attribute addProperty Name "Status_of_input_A"}
    Status_of_input_A : BOOL;
    {attribute addProperty Name "Status_of_input_B"}
    Status_of_input_B : BOOL;
    {attribute addProperty Name "Status_of_input_C"}
    Status_of_input_C : BOOL;
    {attribute addProperty Name "Status_of_extern_latch"}
    Status_of_extern_latch : BOOL;
    {attribute addProperty Name "Sync_error"}
    Sync_error : BOOL;
    {attribute addProperty Name "TxPDO_Toggle"}
    TxPDO_Toggle : BOOL;
END_STRUCT
END_TYPE

// ---- DUTs/IO/PdoEntries/Control_6EF2C5D0.TcDUT
{attribute 'GeneratedUsingTerminal: EL7041-1000-0021'}
{attribute addProperty BoxType "EL7041-1000-0021"}
{attribute addProperty Id "Enable_latch_CBOOL1Enable_latch_extern_on_positive_edgeBOOL1Set_counterBOOL1Enable_latch_extern_on_negative_edgeBOOL1"}
{attribute addProperty CRC "1861404112"}
{attribute addProperty Size "4"}
TYPE Control_6EF2C5D0 :
STRUCT
    {attribute addProperty Name "Enable_latch_C"}
    Enable_latch_C : BOOL;
    {attribute addProperty Name "Enable_latch_extern_on_positive_edge"}
    Enable_latch_extern_on_positive_edge : BOOL;
    {attribute addProperty Name "Set_counter"}
    Set_counter : BOOL;
    {attribute addProperty Name "Enable_latch_extern_on_negative_edge"}
    Enable_latch_extern_on_negative_edge : BOOL;
END_STRUCT
END_TYPE

// ---- DUTs/IO/PDOs/COM_TxPDO_Map_Inputs_Channel_3801C95E.TcDUT
{attribute 'GeneratedUsingTerminal: EL6002-0000-0019'}
{attribute addProperty BoxType "EL6002-0000-0019"}
{attribute addProperty Id "StatusAT %I*Status_3D84275F8Data_InAT %I*ARRAY[0..21] OF USINT22"}
{attribute addProperty CRC "1334739266"}
{attribute addProperty Size "30"}
TYPE COM_TxPDO_Map_Inputs_Channel_3801C95E EXTENDS TcoIo.InputBase_8311D824 :
STRUCT
    {attribute addProperty Name "Status"}
    Status AT %I* : Status_3D84275F;
    {attribute addProperty Name "Data_In"}
    Data_In AT %I* : ARRAY[0..21] OF USINT;
END_STRUCT
END_TYPE

// ---- DUTs/IO/PDOs/COM_RxPDO_Map_Outputs_Channel_EADA2E0D.TcDUT
{attribute 'GeneratedUsingTerminal: EL6002-0000-0019'}
{attribute addProperty BoxType "EL6002-0000-0019"}
{attribute addProperty Id "CtrlAT %Q*Ctrl_1EFB4D3B5Data_OutAT %Q*ARRAY[0..21] OF USINT22"}
{attribute addProperty CRC "3494673196"}
{attribute addProperty Size "27"}
TYPE COM_RxPDO_Map_Outputs_Channel_EADA2E0D EXTENDS TcoIo.OutputBase_10CEE7DE :
STRUCT
    {attribute addProperty Name "Ctrl"}
    Ctrl AT %Q* : Ctrl_1EFB4D3B;
    {attribute addProperty Name "Data_Out"}
    Data_Out AT %Q* : ARRAY[0..21] OF USINT;
END_STRUCT
END_TYPE

// ---- DUTs/IO/PDOs/Channel_830843C1.TcDUT
{attribute 'GeneratedUsingTerminal: EL1809-0000-0018'}
{attribute addProperty BoxType "EL1809-0000-0018"}
{attribute addProperty Id "InputAT %I*BOOL1"}
{attribute addProperty CRC "2198356929"}
{attribute addProperty Size "1"}
TYPE Channel_830843C1 EXTENDS TcoIo.InputBase_8311D824 :
STRUCT
    {attribute addProperty Name "Input"}
    Input AT %I* : BOOL;
END_STRUCT
END_TYPE

// ---- DUTs/IO/PDOs/Channel_42CA91F7.TcDUT
{attribute 'GeneratedUsingTerminal: EL2809-0000-0018'}
{attribute addProperty BoxType "EL2809-0000-0018"}
{attribute addProperty Id "OutputAT %Q*BOOL1"}
{attribute addProperty CRC "1120571895"}
{attribute addProperty Size "1"}
TYPE Channel_42CA91F7 EXTENDS TcoIo.OutputBase_10CEE7DE :
STRUCT
    {attribute addProperty Name "Output"}
    Output AT %Q* : BOOL;
END_STRUCT
END_TYPE

// ---- DUTs/IO/PDOs/AO_Output_Channel_BA7EBB7C.TcDUT
{attribute 'GeneratedUsingTerminal: EL4004-0000-0020'}
{attribute addProperty BoxType "EL4004-0000-0020"}
{attribute addProperty Id "Analog_outputAT %Q*INT2"}
{attribute addProperty CRC "3128867708"}
{attribute addProperty Size "2"}
TYPE AO_Output_Channel_BA7EBB7C EXTENDS TcoIo.OutputBase_10CEE7DE :
STRUCT
    {attribute addProperty Name "Analog_output"}
    Analog_output AT %Q* : INT;
END_STRUCT
END_TYPE

// ---- DUTs/IO/PDOs/COM_Inputs_3801C95E.TcDUT
{attribute 'GeneratedUsingTerminal: EL6001-0000-0020'}
{attribute addProperty BoxType "EL6001-0000-0020"}
{attribute addProperty Id "StatusAT %I*Status_3D84275F8Data_InAT %I*ARRAY[0..21] OF USINT22"}
{attribute addProperty CRC "1334739266"}
{attribute addProperty Size "30"}
TYPE COM_Inputs_3801C95E EXTENDS TcoIo.InputBase_8311D824 :
STRUCT
    {attribute addProperty Name "Status"}
    Status AT %I* : Status_3D84275F;
    {attribute addProperty Name "Data_In"}
    Data_In AT %I* : ARRAY[0..21] OF USINT;
END_STRUCT
END_TYPE

// ---- DUTs/IO/PDOs/COM_Outputs_DEF408EC.TcDUT
{attribute 'GeneratedUsingTerminal: EL6001-0000-0020'}
{attribute addProperty BoxType "EL6001-0000-0020"}
{attribute addProperty Id "CtrlAT %Q*Ctrl_71604E865Data_OutAT %Q*ARRAY[0..21] OF USINT22"}
{attribute addProperty CRC "2695605661"}
{attribute addProperty Size "27"}
TYPE COM_Outputs_DEF408EC EXTENDS TcoIo.OutputBase_10CEE7DE :
STRUCT
    {attribute addProperty Name "Ctrl"}
    Ctrl AT %Q* : Ctrl_71604E86;
    {attribute addProperty Name "Data_Out"}
    Data_Out AT %Q* : ARRAY[0..21] OF USINT;
END_STRUCT
END_TYPE

// ---- DUTs/IO/PDOs/AI_Standard_Channel_A8DF64E3.TcDUT
{attribute 'GeneratedUsingTerminal: EL3174-0002-0017'}
{attribute addProperty BoxType "EL3174-0002-0017"}
{attribute addProperty Id "StatusAT %I*Status_B07533568ValueAT %I*INT2"}
{attribute addProperty CRC "2833212643"}
{attribute addProperty Size "10"}
TYPE AI_Standard_Channel_A8DF64E3 EXTENDS TcoIo.InputBase_8311D824 :
STRUCT
    {attribute addProperty Name "Status"}
    Status AT %I* : Status_B0753356;
    {attribute addProperty Name "Value"}
    Value AT %I* : INT;
END_STRUCT
END_TYPE

// ---- DUTs/IO/PDOs/AI_Standard_Channel_4A394481.TcDUT
{attribute 'GeneratedUsingTerminal: EL3011-0000-0018'}
{attribute addProperty BoxType "EL3011-0000-0018"}
{attribute addProperty Id "StatusAT %I*Status_F2CE6D917ValueAT %I*INT2"}
{attribute addProperty CRC "1245267073"}
{attribute addProperty Size "9"}
TYPE AI_Standard_Channel_4A394481 EXTENDS TcoIo.InputBase_8311D824 :
STRUCT
    {attribute addProperty Name "Status"}
    Status AT %I* : Status_F2CE6D91;
    {attribute addProperty Name "Value"}
    Value AT %I* : INT;
END_STRUCT
END_TYPE

// ---- DUTs/IO/PDOs/L1_Voltage_Status_7371B043.TcDUT
{attribute 'GeneratedUsingTerminal: EL3773-0000-0021'}
{attribute addProperty BoxType "EL3773-0000-0021"}
{attribute addProperty Id "U1_StatusAT %I*U1_Status_DC9039207"}
{attribute addProperty CRC "1936830531"}
{attribute addProperty Size "7"}
TYPE L1_Voltage_Status_7371B043 EXTENDS TcoIo.InputBase_8311D824 :
STRUCT
    {attribute addProperty Name "U1_Status"}
    U1_Status AT %I* : U1_Status_DC903920;
END_STRUCT
END_TYPE

// ---- DUTs/IO/PDOs/L1_Voltage_Samples_41AEB7FF.TcDUT
{attribute 'GeneratedUsingTerminal: EL3773-0000-0021'}
{attribute addProperty BoxType "EL3773-0000-0021"}
{attribute addProperty Id "U1_SamplesAT %I*U1_Samples_2549228720"}
{attribute addProperty CRC "1101969407"}
{attribute addProperty Size "20"}
TYPE L1_Voltage_Samples_41AEB7FF EXTENDS TcoIo.InputBase_8311D824 :
STRUCT
    {attribute addProperty Name "U1_Samples"}
    U1_Samples AT %I* : U1_Samples_25492287;
END_STRUCT
END_TYPE

// ---- DUTs/IO/PDOs/L1_Current_Status_82DECBF6.TcDUT
{attribute 'GeneratedUsingTerminal: EL3773-0000-0021'}
{attribute addProperty BoxType "EL3773-0000-0021"}
{attribute addProperty Id "I1_StatusAT %I*I1_Status_DC9039207"}
{attribute addProperty CRC "2195639286"}
{attribute addProperty Size "7"}
TYPE L1_Current_Status_82DECBF6 EXTENDS TcoIo.InputBase_8311D824 :
STRUCT
    {attribute addProperty Name "I1_Status"}
    I1_Status AT %I* : I1_Status_DC903920;
END_STRUCT
END_TYPE

// ---- DUTs/IO/PDOs/L1_Current_Samples_9EC08B3E.TcDUT
{attribute 'GeneratedUsingTerminal: EL3773-0000-0021'}
{attribute addProperty BoxType "EL3773-0000-0021"}
{attribute addProperty Id "I1_SamplesAT %I*I1_Samples_2549228720"}
{attribute addProperty CRC "2663418686"}
{attribute addProperty Size "20"}
TYPE L1_Current_Samples_9EC08B3E EXTENDS TcoIo.InputBase_8311D824 :
STRUCT
    {attribute addProperty Name "I1_Samples"}
    I1_Samples AT %I* : I1_Samples_25492287;
END_STRUCT
END_TYPE

// ---- DUTs/IO/PDOs/L2_Voltage_Status_0D1813FE.TcDUT
{attribute 'GeneratedUsingTerminal: EL3773-0000-0021'}
{attribute addProperty BoxType "EL3773-0000-0021"}
{attribute addProperty Id "U2_StatusAT %I*U2_Status_DC9039207"}
{attribute addProperty CRC "219681790"}
{attribute addProperty Size "7"}
TYPE L2_Voltage_Status_0D1813FE EXTENDS TcoIo.InputBase_8311D824 :
STRUCT
    {attribute addProperty Name "U2_Status"}
    U2_Status AT %I* : U2_Status_DC903920;
END_STRUCT
END_TYPE

// ---- DUTs/IO/PDOs/L2_Voltage_Samples_75D833AF.TcDUT
{attribute 'GeneratedUsingTerminal: EL3773-0000-0021'}
{attribute addProperty BoxType "EL3773-0000-0021"}
{attribute addProperty Id "U2_SamplesAT %I*U2_Samples_2549228720"}
{attribute addProperty CRC "1977103279"}
{attribute addProperty Size "20"}
TYPE L2_Voltage_Samples_75D833AF EXTENDS TcoIo.InputBase_8311D824 :
STRUCT
    {attribute addProperty Name "U2_Samples"}
    U2_Samples AT %I* : U2_Samples_25492287;
END_STRUCT
END_TYPE

// ---- DUTs/IO/PDOs/L2_Current_Status_FCB7684B.TcDUT
{attribute 'GeneratedUsingTerminal: EL3773-0000-0021'}
{attribute addProperty BoxType "EL3773-0000-0021"}
{attribute addProperty Id "I2_StatusAT %I*I2_Status_DC9039207"}
{attribute addProperty CRC "4239878219"}
{attribute addProperty Size "7"}
TYPE L2_Current_Status_FCB7684B EXTENDS TcoIo.InputBase_8311D824 :
STRUCT
    {attribute addProperty Name "I2_Status"}
    I2_Status AT %I* : I2_Status_DC903920;
END_STRUCT
END_TYPE

// ---- DUTs/IO/PDOs/L2_Current_Samples_AAB60F6E.TcDUT
{attribute 'GeneratedUsingTerminal: EL3773-0000-0021'}
{attribute addProperty BoxType "EL3773-0000-0021"}
{attribute addProperty Id "I2_SamplesAT %I*I2_Samples_2549228720"}
{attribute addProperty CRC "2864058222"}
{attribute addProperty Size "20"}
TYPE L2_Current_Samples_AAB60F6E EXTENDS TcoIo.InputBase_8311D824 :
STRUCT
    {attribute addProperty Name "I2_Samples"}
    I2_Samples AT %I* : I2_Samples_25492287;
END_STRUCT
END_TYPE

// ---- DUTs/IO/PDOs/L3_Voltage_Status_273F7295.TcDUT
{attribute 'GeneratedUsingTerminal: EL3773-0000-0021'}
{attribute addProperty BoxType "EL3773-0000-0021"}
{attribute addProperty Id "U3_StatusAT %I*U3_Status_DC9039207"}
{attribute addProperty CRC "658469525"}
{attribute addProperty Size "7"}
TYPE L3_Voltage_Status_273F7295 EXTENDS TcoIo.InputBase_8311D824 :
STRUCT
    {attribute addProperty Name "U3_Status"}
    U3_Status AT %I* : U3_Status_DC903920;
END_STRUCT
END_TYPE

// ---- DUTs/IO/PDOs/L3_Voltage_Samples_660A4F9F.TcDUT
{attribute 'GeneratedUsingTerminal: EL3773-0000-0021'}
{attribute addProperty BoxType "EL3773-0000-0021"}
{attribute addProperty Id "U3_SamplesAT %I*U3_Samples_2549228720"}
{attribute addProperty CRC "1711951775"}
{attribute addProperty Size "20"}
TYPE L3_Voltage_Samples_660A4F9F EXTENDS TcoIo.InputBase_8311D824 :
STRUCT
    {attribute addProperty Name "U3_Samples"}
    U3_Samples AT %I* : U3_Samples_25492287;
END_STRUCT
END_TYPE

// ---- DUTs/IO/PDOs/L3_Current_Status_D6900920.TcDUT
{attribute 'GeneratedUsingTerminal: EL3773-0000-0021'}
{attribute addProperty BoxType "EL3773-0000-0021"}
{attribute addProperty Id "I3_StatusAT %I*I3_Status_DC9039207"}
{attribute addProperty CRC "3599763744"}
{attribute addProperty Size "7"}
TYPE L3_Current_Status_D6900920 EXTENDS TcoIo.InputBase_8311D824 :
STRUCT
    {attribute addProperty Name "I3_Status"}
    I3_Status AT %I* : I3_Status_DC903920;
END_STRUCT
END_TYPE

// ---- DUTs/IO/PDOs/L3_Current_Samples_B964735E.TcDUT
{attribute 'GeneratedUsingTerminal: EL3773-0000-0021'}
{attribute addProperty BoxType "EL3773-0000-0021"}
{attribute addProperty Id "I3_SamplesAT %I*I3_Samples_2549228720"}
{attribute addProperty CRC "3110368094"}
{attribute addProperty Size "20"}
TYPE L3_Current_Samples_B964735E EXTENDS TcoIo.InputBase_8311D824 :
STRUCT
    {attribute addProperty Name "I3_Samples"}
    I3_Samples AT %I* : I3_Samples_25492287;
END_STRUCT
END_TYPE

// ---- DUTs/IO/PDOs/AI_NextSync1Time_6DC4D296.TcDUT
{attribute 'GeneratedUsingTerminal: EL3773-0000-0021'}
{attribute addProperty BoxType "EL3773-0000-0021"}
{attribute addProperty Id "StartTimeNextLatchAT %I*StartTimeNextLatch_02E0C1C88"}
{attribute addProperty CRC "1841615510"}
{attribute addProperty Size "8"}
TYPE AI_NextSync1Time_6DC4D296 EXTENDS TcoIo.InputBase_8311D824 :
STRUCT
    {attribute addProperty Name "StartTimeNextLatch"}
    StartTimeNextLatch AT %I* : StartTimeNextLatch_02E0C1C8;
END_STRUCT
END_TYPE

// ---- DUTs/IO/PDOs/AI_Sample_Count_EA88CAD9.TcDUT
{attribute 'GeneratedUsingTerminal: EL3773-0000-0021'}
{attribute addProperty BoxType "EL3773-0000-0021"}
{attribute addProperty Id "Sample_CountAT %I*UINT2"}
{attribute addProperty CRC "3934833369"}
{attribute addProperty Size "2"}
TYPE AI_Sample_Count_EA88CAD9 EXTENDS TcoIo.InputBase_8311D824 :
STRUCT
    {attribute addProperty Name "Sample_Count"}
    Sample_Count AT %I* : UINT;
END_STRUCT
END_TYPE

// ---- DUTs/IO/PDOs/InfoData_B84DBEC5.TcDUT
{attribute 'GeneratedUsingTerminal: EL3773-0000-0021'}
{attribute addProperty BoxType "EL3773-0000-0021"}
{attribute addProperty Id "AdsAddrAT %I*TcoIo.TcoAmsAddr0DcOutputShiftAT %I*DINT4DcInputShiftAT %I*DINT4StateAT %I*UINT2"}
{attribute addProperty CRC "3092102853"}
{attribute addProperty Size "10"}
TYPE InfoData_B84DBEC5 EXTENDS TcoIo.InputBase_8311D824 :
STRUCT
    {attribute addProperty Name "AdsAddr"}
    AdsAddr AT %I* : TcoIo.TcoAmsAddr;
    {attribute addProperty Name "DcOutputShift"}
    DcOutputShift AT %I* : DINT;
    {attribute addProperty Name "DcInputShift"}
    DcInputShift AT %I* : DINT;
    {attribute addProperty Name "State"}
    State AT %I* : UINT;
END_STRUCT
END_TYPE

// ---- DUTs/IO/PDOs/MTO_Inputs_Channel_53C09E8B.TcDUT
{attribute 'GeneratedUsingTerminal: EL2258-0000-0017'}
{attribute addProperty BoxType "EL2258-0000-0017"}
{attribute addProperty Id "StatusAT %I*Status_642C2ED16"}
{attribute addProperty CRC "1405132427"}
{attribute addProperty Size "6"}
TYPE MTO_Inputs_Channel_53C09E8B EXTENDS TcoIo.InputBase_8311D824 :
STRUCT
    {attribute addProperty Name "Status"}
    Status AT %I* : Status_642C2ED1;
END_STRUCT
END_TYPE

// ---- DUTs/IO/PDOs/MTO_Outputs_10x_Channel_A3C0C022.TcDUT
{attribute 'GeneratedUsingTerminal: EL2258-0000-0017'}
{attribute addProperty BoxType "EL2258-0000-0017"}
{attribute addProperty Id "CtrlAT %Q*Ctrl_77460BD36OutputsAT %Q*Outputs_A910484D10Output_event_timeAT %Q*ARRAY[0..9] OF UDINT40"}
{attribute addProperty CRC "922776817"}
{attribute addProperty Size "56"}
TYPE MTO_Outputs_10x_Channel_A3C0C022 EXTENDS TcoIo.OutputBase_10CEE7DE :
STRUCT
    {attribute addProperty Name "Ctrl"}
    Ctrl AT %Q* : Ctrl_77460BD3;
    {attribute addProperty Name "Outputs"}
    Outputs AT %Q* : Outputs_A910484D;
    {attribute addProperty Name "Output_event_time"}
    Output_event_time AT %Q* : ARRAY[0..9] OF UDINT;
END_STRUCT
END_TYPE

// ---- DUTs/IO/PDOs/PM_Inputs_Channel_2F868086.TcDUT
{attribute 'GeneratedUsingTerminal: EL3403-0000-0023'}
{attribute addProperty BoxType "EL3403-0000-0023"}
{attribute addProperty Id "TxPDO_ToggleAT %I*BOOL1CurrentAT %I*DINT4VoltageAT %I*DINT4Active_powerAT %I*DINT4IndexAT %I*USINT1Variant_valueAT %I*DINT4"}
{attribute addProperty CRC "797343878"}
{attribute addProperty Size "18"}
TYPE PM_Inputs_Channel_2F868086 EXTENDS TcoIo.InputBase_8311D824 :
STRUCT
    {attribute addProperty Name "TxPDO_Toggle"}
    TxPDO_Toggle AT %I* : BOOL;
    {attribute addProperty Name "Current"}
    Current AT %I* : DINT;
    {attribute addProperty Name "Voltage"}
    Voltage AT %I* : DINT;
    {attribute addProperty Name "Active_power"}
    Active_power AT %I* : DINT;
    {attribute addProperty Name "Index"}
    Index AT %I* : USINT;
    {attribute addProperty Name "Variant_value"}
    Variant_value AT %I* : DINT;
END_STRUCT
END_TYPE

// ---- DUTs/IO/PDOs/PM_Status_data_2A9514CB.TcDUT
{attribute 'GeneratedUsingTerminal: EL3403-0000-0023'}
{attribute addProperty BoxType "EL3403-0000-0023"}
{attribute addProperty Id "Missing_zero_crossing_AAT %I*BOOL1Missing_zero_crossing_BAT %I*BOOL1Missing_zero_crossing_CAT %I*BOOL1Phase_sequence_errorAT %I*BOOL1"}
{attribute addProperty CRC "714413259"}
{attribute addProperty Size "4"}
TYPE PM_Status_data_2A9514CB EXTENDS TcoIo.InputBase_8311D824 :
STRUCT
    {attribute addProperty Name "Missing_zero_crossing_A"}
    Missing_zero_crossing_A AT %I* : BOOL;
    {attribute addProperty Name "Missing_zero_crossing_B"}
    Missing_zero_crossing_B AT %I* : BOOL;
    {attribute addProperty Name "Missing_zero_crossing_C"}
    Missing_zero_crossing_C AT %I* : BOOL;
    {attribute addProperty Name "Phase_sequence_error"}
    Phase_sequence_error AT %I* : BOOL;
END_STRUCT
END_TYPE

// ---- DUTs/IO/PDOs/PM_Outputs_Channel_E5FBDE30.TcDUT
{attribute 'GeneratedUsingTerminal: EL3403-0000-0023'}
{attribute addProperty BoxType "EL3403-0000-0023"}
{attribute addProperty Id "IndexAT %Q*USINT1"}
{attribute addProperty CRC "3858488880"}
{attribute addProperty Size "1"}
TYPE PM_Outputs_Channel_E5FBDE30 EXTENDS TcoIo.OutputBase_10CEE7DE :
STRUCT
    {attribute addProperty Name "Index"}
    Index AT %Q* : USINT;
END_STRUCT
END_TYPE

// ---- DUTs/IO/PDOs/AT_x_4EC2E768.TcDUT
{attribute 'GeneratedUsingTerminal: AX5101-0000-0214-0214'}
{attribute addProperty BoxType "AX5101-0000-0214-0214"}
{attribute addProperty Id "Drive_status_wordAT %I*UINT2Position_feedback_1_valueAT %I*DINT4Following_distanceAT %I*DINT4"}
{attribute addProperty CRC "1321396072"}
{attribute addProperty Size "10"}
TYPE AT_x_4EC2E768 EXTENDS TcoIo.InputBase_8311D824 :
STRUCT
    {attribute addProperty Name "Drive_status_word"}
    Drive_status_word AT %I* : UINT;
    {attribute addProperty Name "Position_feedback_1_value"}
    Position_feedback_1_value AT %I* : DINT;
    {attribute addProperty Name "Following_distance"}
    Following_distance AT %I* : DINT;
END_STRUCT
END_TYPE

// ---- DUTs/IO/PDOs/MDT_864618EC.TcDUT
{attribute 'GeneratedUsingTerminal: AX5101-0000-0214-0214'}
{attribute addProperty BoxType "AX5101-0000-0214-0214"}
{attribute addProperty Id "Master_control_wordAT %Q*UINT2Position_command_valueAT %Q*DINT4"}
{attribute addProperty CRC "2252740844"}
{attribute addProperty Size "6"}
TYPE MDT_864618EC EXTENDS TcoIo.OutputBase_10CEE7DE :
STRUCT
    {attribute addProperty Name "Master_control_word"}
    Master_control_word AT %Q* : UINT;
    {attribute addProperty Name "Position_command_value"}
    Position_command_value AT %Q* : DINT;
END_STRUCT
END_TYPE

// ---- DUTs/IO/PDOs/InfoData_F60A43AC.TcDUT
{attribute 'GeneratedUsingTerminal: AX5101-0000-0214-0214'}
{attribute addProperty BoxType "AX5101-0000-0214-0214"}
{attribute addProperty Id "AdsAddrAT %I*TcoIo.TcoAmsAddr0DcOutputShiftAT %I*DINT4DcInputShiftAT %I*DINT4Chn0AT %I*USINT1StateAT %I*UINT2"}
{attribute addProperty CRC "4127867820"}
{attribute addProperty Size "11"}
TYPE InfoData_F60A43AC EXTENDS TcoIo.InputBase_8311D824 :
STRUCT
    {attribute addProperty Name "AdsAddr"}
    AdsAddr AT %I* : TcoIo.TcoAmsAddr;
    {attribute addProperty Name "DcOutputShift"}
    DcOutputShift AT %I* : DINT;
    {attribute addProperty Name "DcInputShift"}
    DcInputShift AT %I* : DINT;
    {attribute addProperty Name "Chn0"}
    Chn0 AT %I* : USINT;
    {attribute addProperty Name "State"}
    State AT %I* : UINT;
END_STRUCT
END_TYPE

// ---- DUTs/IO/PDOs/Device_State_B9CC7757.TcDUT
{attribute 'GeneratedUsingTerminal: AES-D-BC-ECAT-0000'}
{attribute addProperty BoxType "AES-D-BC-ECAT-0000"}
{attribute addProperty Id "CouplerStateAT %I*UDINT4"}
{attribute addProperty CRC "3117184855"}
{attribute addProperty Size "4"}
TYPE Device_State_B9CC7757 EXTENDS TcoIo.InputBase_8311D824 :
STRUCT
    {attribute addProperty Name "CouplerState"}
    CouplerState AT %I* : UDINT;
END_STRUCT
END_TYPE

// ---- DUTs/IO/PDOs/Device_Control_33EFE70E.TcDUT
{attribute 'GeneratedUsingTerminal: AES-D-BC-ECAT-0000'}
{attribute addProperty BoxType "AES-D-BC-ECAT-0000"}
{attribute addProperty Id "CouplerCtrlAT %Q*UDINT4"}
{attribute addProperty CRC "871360270"}
{attribute addProperty Size "4"}
TYPE Device_Control_33EFE70E EXTENDS TcoIo.OutputBase_10CEE7DE :
STRUCT
    {attribute addProperty Name "CouplerCtrl"}
    CouplerCtrl AT %Q* : UDINT;
END_STRUCT
END_TYPE

// ---- DUTs/IO/PDOs/Inputs_03C60166.TcDUT
{attribute 'GeneratedUsingTerminal: AES-D-BC-ECAT-0000'}
{attribute addProperty BoxType "AES-D-BC-ECAT-0000"}
{attribute addProperty Id "digital_Data_IAT %I*ARRAY[0..27] OF USINT28"}
{attribute addProperty CRC "2446583242"}
{attribute addProperty Size "28"}
TYPE Inputs_03C60166 EXTENDS TcoIo.InputBase_8311D824 :
STRUCT
    {attribute addProperty Name "digital_Data_I"}
    digital_Data_I AT %I* : ARRAY[0..27] OF USINT;
END_STRUCT
END_TYPE

// ---- DUTs/IO/PDOs/Outputs_79BC345B.TcDUT
{attribute 'GeneratedUsingTerminal: AES-D-BC-ECAT-0000'}
{attribute addProperty BoxType "AES-D-BC-ECAT-0000"}
{attribute addProperty Id "digital_Data_OAT %Q*ARRAY[0..27] OF USINT28"}
{attribute addProperty CRC "3096397179"}
{attribute addProperty Size "28"}
TYPE Outputs_79BC345B EXTENDS TcoIo.OutputBase_10CEE7DE :
STRUCT
    {attribute addProperty Name "digital_Data_O"}
    digital_Data_O AT %Q* : ARRAY[0..27] OF USINT;
END_STRUCT
END_TYPE

// ---- DUTs/IO/PDOs/Module_1_32_Byte_Valve_Unit_0x7F_1A3DA03C.TcDUT
{attribute 'GeneratedUsingTerminal: AES-D-BC-ECAT-0000'}
{attribute addProperty BoxType "AES-D-BC-ECAT-0000"}
{attribute addProperty Id "InputsInputs_03C6016628OutputsOutputs_79BC345B28"}
{attribute addProperty CRC "440246332"}
{attribute addProperty Size "56"}
TYPE Module_1_32_Byte_Valve_Unit_0x7F_1A3DA03C :
STRUCT
    {attribute addProperty Name "Inputs"}
    Inputs : Inputs_03C60166;
    {attribute addProperty Name "Outputs"}
    Outputs : Outputs_79BC345B;
END_STRUCT
END_TYPE

// ---- DUTs/IO/PDOs/InfoData_8F85596B.TcDUT
{attribute 'GeneratedUsingTerminal: EL6631-0000-0018'}
{attribute addProperty BoxType "EL6631-0000-0018"}
{attribute addProperty Id "AdsAddrAT %I*TcoIo.TcoAmsAddr0AoeNetIdAT %I*TcoIo.TcoAmsNetId0StateAT %I*UINT2"}
{attribute addProperty CRC "2407881067"}
{attribute addProperty Size "2"}
TYPE InfoData_8F85596B EXTENDS TcoIo.InputBase_8311D824 :
STRUCT
    {attribute addProperty Name "AdsAddr"}
    AdsAddr AT %I* : TcoIo.TcoAmsAddr;
    {attribute addProperty Name "AoeNetId"}
    AoeNetId AT %I* : TcoIo.TcoAmsNetId;
    {attribute addProperty Name "State"}
    State AT %I* : UINT;
END_STRUCT
END_TYPE

// ---- DUTs/IO/PDOs/Device_State_384275F8.TcDUT
{attribute 'GeneratedUsingTerminal: AES-D-BC-ECAT-0000'}
{attribute addProperty BoxType "AES-D-BC-ECAT-0000"}
{attribute addProperty Id "IO_1_8AT %I*BYTE1IO_9_10AT %I*BYTE1ValveExtSupplyDiag_1_6AT %I*BYTE1SupplyAT %I*BYTE1CommonValveAT %I*BOOL1ConfigDiagnosisLAT %I*BYTE1Switch_Count_StoredAT %I*BOOL1Heardbeat_xAT %I*BOOL1ConfigDiagnosisHAT %I*BYTE1"}
{attribute addProperty CRC "943879672"}
{attribute addProperty Size "9"}
TYPE Device_State_384275F8 EXTENDS TcoIo.InputBase_8311D824 :
STRUCT
    {attribute addProperty Name "IO_1_8"}
    IO_1_8 AT %I* : BYTE;
    {attribute addProperty Name "IO_9_10"}
    IO_9_10 AT %I* : BYTE;
    {attribute addProperty Name "ValveExtSupplyDiag_1_6"}
    ValveExtSupplyDiag_1_6 AT %I* : BYTE;
    {attribute addProperty Name "Supply"}
    Supply AT %I* : BYTE;
    {attribute addProperty Name "CommonValve"}
    CommonValve AT %I* : BOOL;
    {attribute addProperty Name "ConfigDiagnosisL"}
    ConfigDiagnosisL AT %I* : BYTE;
    {attribute addProperty Name "Switch_Count_Stored"}
    Switch_Count_Stored AT %I* : BOOL;
    {attribute addProperty Name "Heardbeat_x"}
    Heardbeat_x AT %I* : BOOL;
    {attribute addProperty Name "ConfigDiagnosisH"}
    ConfigDiagnosisH AT %I* : BYTE;
END_STRUCT
END_TYPE

// ---- DUTs/IO/PDOs/Device_Control_5857DF0F.TcDUT
{attribute 'GeneratedUsingTerminal: AES-D-BC-ECAT-0000'}
{attribute addProperty BoxType "AES-D-BC-ECAT-0000"}
{attribute addProperty Id "Switch_Count_StoreAT %Q*BOOL1HL_SwapAT %Q*BOOL1Default_Modul_ControlAT %Q*BOOL1"}
{attribute addProperty CRC "1482153743"}
{attribute addProperty Size "3"}
TYPE Device_Control_5857DF0F EXTENDS TcoIo.OutputBase_10CEE7DE :
STRUCT
    {attribute addProperty Name "Switch_Count_Store"}
    Switch_Count_Store AT %Q* : BOOL;
    {attribute addProperty Name "HL_Swap"}
    HL_Swap AT %Q* : BOOL;
    {attribute addProperty Name "Default_Modul_Control"}
    Default_Modul_Control AT %Q* : BOOL;
END_STRUCT
END_TYPE

// ---- DUTs/IO/PDOs/Inputs_23559BB0.TcDUT
{attribute 'GeneratedUsingTerminal: AES-D-BC-ECAT-0000'}
{attribute addProperty BoxType "AES-D-BC-ECAT-0000"}
{attribute addProperty Id "digital_Data_IAT %I*ARRAY[0..31] OF USINT32"}
{attribute addProperty CRC "1374483313"}
{attribute addProperty Size "32"}
TYPE Inputs_23559BB0 EXTENDS TcoIo.InputBase_8311D824 :
STRUCT
    {attribute addProperty Name "digital_Data_I"}
    digital_Data_I AT %I* : ARRAY[0..31] OF USINT;
END_STRUCT
END_TYPE

// ---- DUTs/IO/PDOs/Outputs_FC2FACAD.TcDUT
{attribute 'GeneratedUsingTerminal: AES-D-BC-ECAT-0000'}
{attribute addProperty BoxType "AES-D-BC-ECAT-0000"}
{attribute addProperty Id "digital_Data_OAT %Q*ARRAY[0..31] OF USINT32"}
{attribute addProperty CRC "2024821696"}
{attribute addProperty Size "32"}
TYPE Outputs_FC2FACAD EXTENDS TcoIo.OutputBase_10CEE7DE :
STRUCT
    {attribute addProperty Name "digital_Data_O"}
    digital_Data_O AT %Q* : ARRAY[0..31] OF USINT;
END_STRUCT
END_TYPE

// ---- DUTs/IO/PDOs/Module_1_32_Byte_Valve_Unit_0x7F_85784B27.TcDUT
{attribute 'GeneratedUsingTerminal: AES-D-BC-ECAT-0000'}
{attribute addProperty BoxType "AES-D-BC-ECAT-0000"}
{attribute addProperty Id "InputsInputs_23559BB032OutputsOutputs_FC2FACAD32"}
{attribute addProperty CRC "2239253287"}
{attribute addProperty Size "64"}
TYPE Module_1_32_Byte_Valve_Unit_0x7F_85784B27 :
STRUCT
    {attribute addProperty Name "Inputs"}
    Inputs : Inputs_23559BB0;
    {attribute addProperty Name "Outputs"}
    Outputs : Outputs_FC2FACAD;
END_STRUCT
END_TYPE

// ---- DUTs/IO/PDOs/DI_TxPDO_Map_DF955083.TcDUT
{attribute 'GeneratedUsingTerminal: IMecat-0007-0001'}
{attribute addProperty BoxType "IMecat-0007-0001"}
{attribute addProperty Id "Pdo_EntryAT %I*ARRAY[0..131] OF USINT132"}
{attribute addProperty CRC "2170192396"}
{attribute addProperty Size "132"}
TYPE DI_TxPDO_Map_DF955083 EXTENDS TcoIo.InputBase_8311D824 :
STRUCT
    {attribute addProperty Name "Pdo_Entry"}
    Pdo_Entry AT %I* : ARRAY[0..131] OF USINT;
END_STRUCT
END_TYPE

// ---- DUTs/IO/PDOs/DO_RxPDO_Map_8BCFF4C9.TcDUT
{attribute 'GeneratedUsingTerminal: IMecat-0007-0001'}
{attribute addProperty BoxType "IMecat-0007-0001"}
{attribute addProperty Id "Pdo_EntryAT %Q*ARRAY[0..33] OF USINT34"}
{attribute addProperty CRC "2035404656"}
{attribute addProperty Size "34"}
TYPE DO_RxPDO_Map_8BCFF4C9 EXTENDS TcoIo.OutputBase_10CEE7DE :
STRUCT
    {attribute addProperty Name "Pdo_Entry"}
    Pdo_Entry AT %Q* : ARRAY[0..33] OF USINT;
END_STRUCT
END_TYPE

// ---- DUTs/IO/PDOs/DCM_Status_Channel_36ED096F.TcDUT
{attribute 'GeneratedUsingTerminal: EL7332-0000-0024'}
{attribute addProperty BoxType "EL7332-0000-0024"}
{attribute addProperty Id "StatusAT %I*Status_B679584511"}
{attribute addProperty CRC "921504111"}
{attribute addProperty Size "11"}
TYPE DCM_Status_Channel_36ED096F EXTENDS TcoIo.InputBase_8311D824 :
STRUCT
    {attribute addProperty Name "Status"}
    Status AT %I* : Status_B6795845;
END_STRUCT
END_TYPE

// ---- DUTs/IO/PDOs/DCM_Synchron_info_data_Channel_6FB37C88.TcDUT
{attribute 'GeneratedUsingTerminal: EL7332-0000-0024'}
{attribute addProperty BoxType "EL7332-0000-0024"}
{attribute addProperty Id "Info_DataAT %I*ARRAY[0..1] OF UINT4"}
{attribute addProperty CRC "1491064414"}
{attribute addProperty Size "4"}
TYPE DCM_Synchron_info_data_Channel_6FB37C88 EXTENDS TcoIo.InputBase_8311D824 :
STRUCT
    {attribute addProperty Name "Info_Data"}
    Info_Data AT %I* : ARRAY[0..1] OF UINT;
END_STRUCT
END_TYPE

// ---- DUTs/IO/PDOs/DCM_Control_Channel_5A8B5016.TcDUT
{attribute 'GeneratedUsingTerminal: EL7332-0000-0024'}
{attribute addProperty BoxType "EL7332-0000-0024"}
{attribute addProperty Id "ControlAT %Q*Control_C948E0F23"}
{attribute addProperty CRC "1519079446"}
{attribute addProperty Size "3"}
TYPE DCM_Control_Channel_5A8B5016 EXTENDS TcoIo.OutputBase_10CEE7DE :
STRUCT
    {attribute addProperty Name "Control"}
    Control AT %Q* : Control_C948E0F2;
END_STRUCT
END_TYPE

// ---- DUTs/IO/PDOs/DCM_Velocity_Channel_A47A3F41.TcDUT
{attribute 'GeneratedUsingTerminal: EL7332-0000-0024'}
{attribute addProperty BoxType "EL7332-0000-0024"}
{attribute addProperty Id "VelocityAT %Q*INT2"}
{attribute addProperty CRC "2759475009"}
{attribute addProperty Size "2"}
TYPE DCM_Velocity_Channel_A47A3F41 EXTENDS TcoIo.OutputBase_10CEE7DE :
STRUCT
    {attribute addProperty Name "Velocity"}
    Velocity AT %Q* : INT;
END_STRUCT
END_TYPE

// ---- DUTs/IO/PDOs/InfoData_F38373C9.TcDUT
{attribute 'GeneratedUsingTerminal: EL7332-0000-0024'}
{attribute addProperty BoxType "EL7332-0000-0024"}
{attribute addProperty Id "AdsAddrAT %I*TcoIo.TcoAmsAddr0Chn0AT %I*USINT1Chn1AT %I*USINT1StateAT %I*UINT2"}
{attribute addProperty CRC "4085478345"}
{attribute addProperty Size "4"}
TYPE InfoData_F38373C9 EXTENDS TcoIo.InputBase_8311D824 :
STRUCT
    {attribute addProperty Name "AdsAddr"}
    AdsAddr AT %I* : TcoIo.TcoAmsAddr;
    {attribute addProperty Name "Chn0"}
    Chn0 AT %I* : USINT;
    {attribute addProperty Name "Chn1"}
    Chn1 AT %I* : USINT;
    {attribute addProperty Name "State"}
    State AT %I* : UINT;
END_STRUCT
END_TYPE

// ---- DUTs/IO/PDOs/Inputs_424E3ECB.TcDUT
{attribute 'GeneratedUsingTerminal: CMMP-AS V4p0 CiA402-0002'}
{attribute addProperty BoxType "CMMP-AS V4p0 CiA402-0002"}
{attribute addProperty Id "StatuswordAT %I*UINT2Mode_Of_Operation_displayAT %I*USINT1Position_Actual_ValueAT %I*DINT4Error_RegisterAT %I*USINT1"}
{attribute addProperty CRC "1112424139"}
{attribute addProperty Size "8"}
TYPE Inputs_424E3ECB EXTENDS TcoIo.InputBase_8311D824 :
STRUCT
    {attribute addProperty Name "Statusword"}
    Statusword AT %I* : UINT;
    {attribute addProperty Name "Mode_Of_Operation_display"}
    Mode_Of_Operation_display AT %I* : USINT;
    {attribute addProperty Name "Position_Actual_Value"}
    Position_Actual_Value AT %I* : DINT;
    {attribute addProperty Name "Error_Register"}
    Error_Register AT %I* : USINT;
END_STRUCT
END_TYPE

// ---- DUTs/IO/PDOs/Inputs_84513182.TcDUT
{attribute 'GeneratedUsingTerminal: CMMP-AS V4p0 CiA402-0002'}
{attribute addProperty BoxType "CMMP-AS V4p0 CiA402-0002"}
{attribute addProperty Id "Velocity_Actual_ValueAT %I*DINT4Following_Error_Actual_ValueAT %I*DINT4"}
{attribute addProperty CRC "2219913602"}
{attribute addProperty Size "8"}
TYPE Inputs_84513182 EXTENDS TcoIo.InputBase_8311D824 :
STRUCT
    {attribute addProperty Name "Velocity_Actual_Value"}
    Velocity_Actual_Value AT %I* : DINT;
    {attribute addProperty Name "Following_Error_Actual_Value"}
    Following_Error_Actual_Value AT %I* : DINT;
END_STRUCT
END_TYPE

// ---- DUTs/IO/PDOs/Outputs_3179CEF4.TcDUT
{attribute 'GeneratedUsingTerminal: CMMP-AS V4p0 CiA402-0002'}
{attribute addProperty BoxType "CMMP-AS V4p0 CiA402-0002"}
{attribute addProperty Id "ControlwordAT %Q*UINT2Mode_Of_OperationAT %Q*USINT1IP_Data_RecordAT %Q*DINT4Homing_MethodAT %Q*SINT1"}
{attribute addProperty CRC "830066420"}
{attribute addProperty Size "8"}
TYPE Outputs_3179CEF4 EXTENDS TcoIo.OutputBase_10CEE7DE :
STRUCT
    {attribute addProperty Name "Controlword"}
    Controlword AT %Q* : UINT;
    {attribute addProperty Name "Mode_Of_Operation"}
    Mode_Of_Operation AT %Q* : USINT;
    {attribute addProperty Name "IP_Data_Record"}
    IP_Data_Record AT %Q* : DINT;
    {attribute addProperty Name "Homing_Method"}
    Homing_Method AT %Q* : SINT;
END_STRUCT
END_TYPE

// ---- DUTs/IO/PDOs/NewMessageFlag_557A079F.TcDUT
{attribute 'GeneratedUsingTerminal: Flexi Gateway GETC1-0001-0000'}
{attribute addProperty BoxType "Flexi Gateway GETC1-0001-0000"}
{attribute addProperty Id "New_Messages_AvailableAT %I*BOOL1"}
{attribute addProperty CRC "1434060703"}
{attribute addProperty Size "1"}
TYPE NewMessageFlag_557A079F EXTENDS TcoIo.InputBase_8311D824 :
STRUCT
    {attribute addProperty Name "New_Messages_Available"}
    New_Messages_Available AT %I* : BOOL;
END_STRUCT
END_TYPE

// ---- DUTs/IO/PDOs/Gateway_to_EtherCAT_Data_100_Bytes_AE1F4D6F.TcDUT
{attribute 'GeneratedUsingTerminal: Flexi Gateway GETC1-0001-0000'}
{attribute addProperty BoxType "Flexi Gateway GETC1-0001-0000"}
{attribute addProperty Id "_100_Bytes_Input_Data_1_4AT %I*ARRAY [0..9] OF BYTE0_100_Bytes_Input_Data_2_4AT %I*ARRAY [0..29] OF BYTE0_100_Bytes_Input_Data_3_4AT %I*ARRAY [0..29] OF BYTE0_100_Bytes_Input_Data_4_4AT %I*ARRAY [0..29] OF BYTE0"}
{attribute addProperty CRC "2921287023"}
{attribute addProperty Size "0"}
TYPE Gateway_to_EtherCAT_Data_100_Bytes_AE1F4D6F EXTENDS TcoIo.InputBase_8311D824 :
STRUCT
    {attribute addProperty Name "_100_Bytes_Input_Data_1_4"}
    _100_Bytes_Input_Data_1_4 AT %I* : ARRAY[0..9] OF BYTE;
    {attribute addProperty Name "_100_Bytes_Input_Data_2_4"}
    _100_Bytes_Input_Data_2_4 AT %I* : ARRAY[0..29] OF BYTE;
    {attribute addProperty Name "_100_Bytes_Input_Data_3_4"}
    _100_Bytes_Input_Data_3_4 AT %I* : ARRAY[0..29] OF BYTE;
    {attribute addProperty Name "_100_Bytes_Input_Data_4_4"}
    _100_Bytes_Input_Data_4_4 AT %I* : ARRAY[0..29] OF BYTE;
END_STRUCT
END_TYPE

// ---- DUTs/IO/PDOs/EtherCAT_to_Gateway_Data_100_Bytes_44CA1D22.TcDUT
{attribute 'GeneratedUsingTerminal: Flexi Gateway GETC1-0001-0000'}
{attribute addProperty BoxType "Flexi Gateway GETC1-0001-0000"}
{attribute addProperty Id "_100_Bytes_Output_Data_1_4AT %Q*ARRAY [0..9] OF BYTE0_100_Bytes_Output_Data_2_4AT %Q*ARRAY [0..29] OF BYTE0_100_Bytes_Output_Data_3_4AT %Q*ARRAY [0..29] OF BYTE0_100_Bytes_Output_Data_4_4AT %Q*ARRAY [0..29] OF BYTE0"}
{attribute addProperty CRC "1154096418"}
{attribute addProperty Size "0"}
TYPE EtherCAT_to_Gateway_Data_100_Bytes_44CA1D22 EXTENDS TcoIo.OutputBase_10CEE7DE :
STRUCT
    {attribute addProperty Name "_100_Bytes_Output_Data_1_4"}
    _100_Bytes_Output_Data_1_4 AT %Q* : ARRAY[0..9] OF BYTE;
    {attribute addProperty Name "_100_Bytes_Output_Data_2_4"}
    _100_Bytes_Output_Data_2_4 AT %Q* : ARRAY[0..29] OF BYTE;
    {attribute addProperty Name "_100_Bytes_Output_Data_3_4"}
    _100_Bytes_Output_Data_3_4 AT %Q* : ARRAY[0..29] OF BYTE;
    {attribute addProperty Name "_100_Bytes_Output_Data_4_4"}
    _100_Bytes_Output_Data_4_4 AT %Q* : ARRAY[0..29] OF BYTE;
END_STRUCT
END_TYPE

// ---- DUTs/IO/PDOs/FB_Position_3FA094ED.TcDUT
{attribute 'GeneratedUsingTerminal: EL7211-0010-0032'}
{attribute addProperty BoxType "EL7211-0010-0032"}
{attribute addProperty Id "PositionAT %I*UDINT4"}
{attribute addProperty CRC "1067488493"}
{attribute addProperty Size "4"}
TYPE FB_Position_3FA094ED EXTENDS TcoIo.InputBase_8311D824 :
STRUCT
    {attribute addProperty Name "Position"}
    Position AT %I* : UDINT;
END_STRUCT
END_TYPE

// ---- DUTs/IO/PDOs/DRV_Statusword_9B36FDFC.TcDUT
{attribute 'GeneratedUsingTerminal: EL7211-0010-0032'}
{attribute addProperty BoxType "EL7211-0010-0032"}
{attribute addProperty Id "StatuswordAT %I*UINT2"}
{attribute addProperty CRC "2604072444"}
{attribute addProperty Size "2"}
TYPE DRV_Statusword_9B36FDFC EXTENDS TcoIo.InputBase_8311D824 :
STRUCT
    {attribute addProperty Name "Statusword"}
    Statusword AT %I* : UINT;
END_STRUCT
END_TYPE

// ---- DUTs/IO/PDOs/DRV_Following_error_actual_value_5AA320BF.TcDUT
{attribute 'GeneratedUsingTerminal: EL7211-0010-0032'}
{attribute addProperty BoxType "EL7211-0010-0032"}
{attribute addProperty Id "Following_error_actual_valueAT %I*DINT4"}
{attribute addProperty CRC "1520640191"}
{attribute addProperty Size "4"}
TYPE DRV_Following_error_actual_value_5AA320BF EXTENDS TcoIo.InputBase_8311D824 :
STRUCT
    {attribute addProperty Name "Following_error_actual_value"}
    Following_error_actual_value AT %I* : DINT;
END_STRUCT
END_TYPE

// ---- DUTs/IO/PDOs/DRV_Controlword_F3F14721.TcDUT
{attribute 'GeneratedUsingTerminal: EL7211-0010-0032'}
{attribute addProperty BoxType "EL7211-0010-0032"}
{attribute addProperty Id "ControlwordAT %Q*UINT2"}
{attribute addProperty CRC "4092675873"}
{attribute addProperty Size "2"}
TYPE DRV_Controlword_F3F14721 EXTENDS TcoIo.OutputBase_10CEE7DE :
STRUCT
    {attribute addProperty Name "Controlword"}
    Controlword AT %Q* : UINT;
END_STRUCT
END_TYPE

